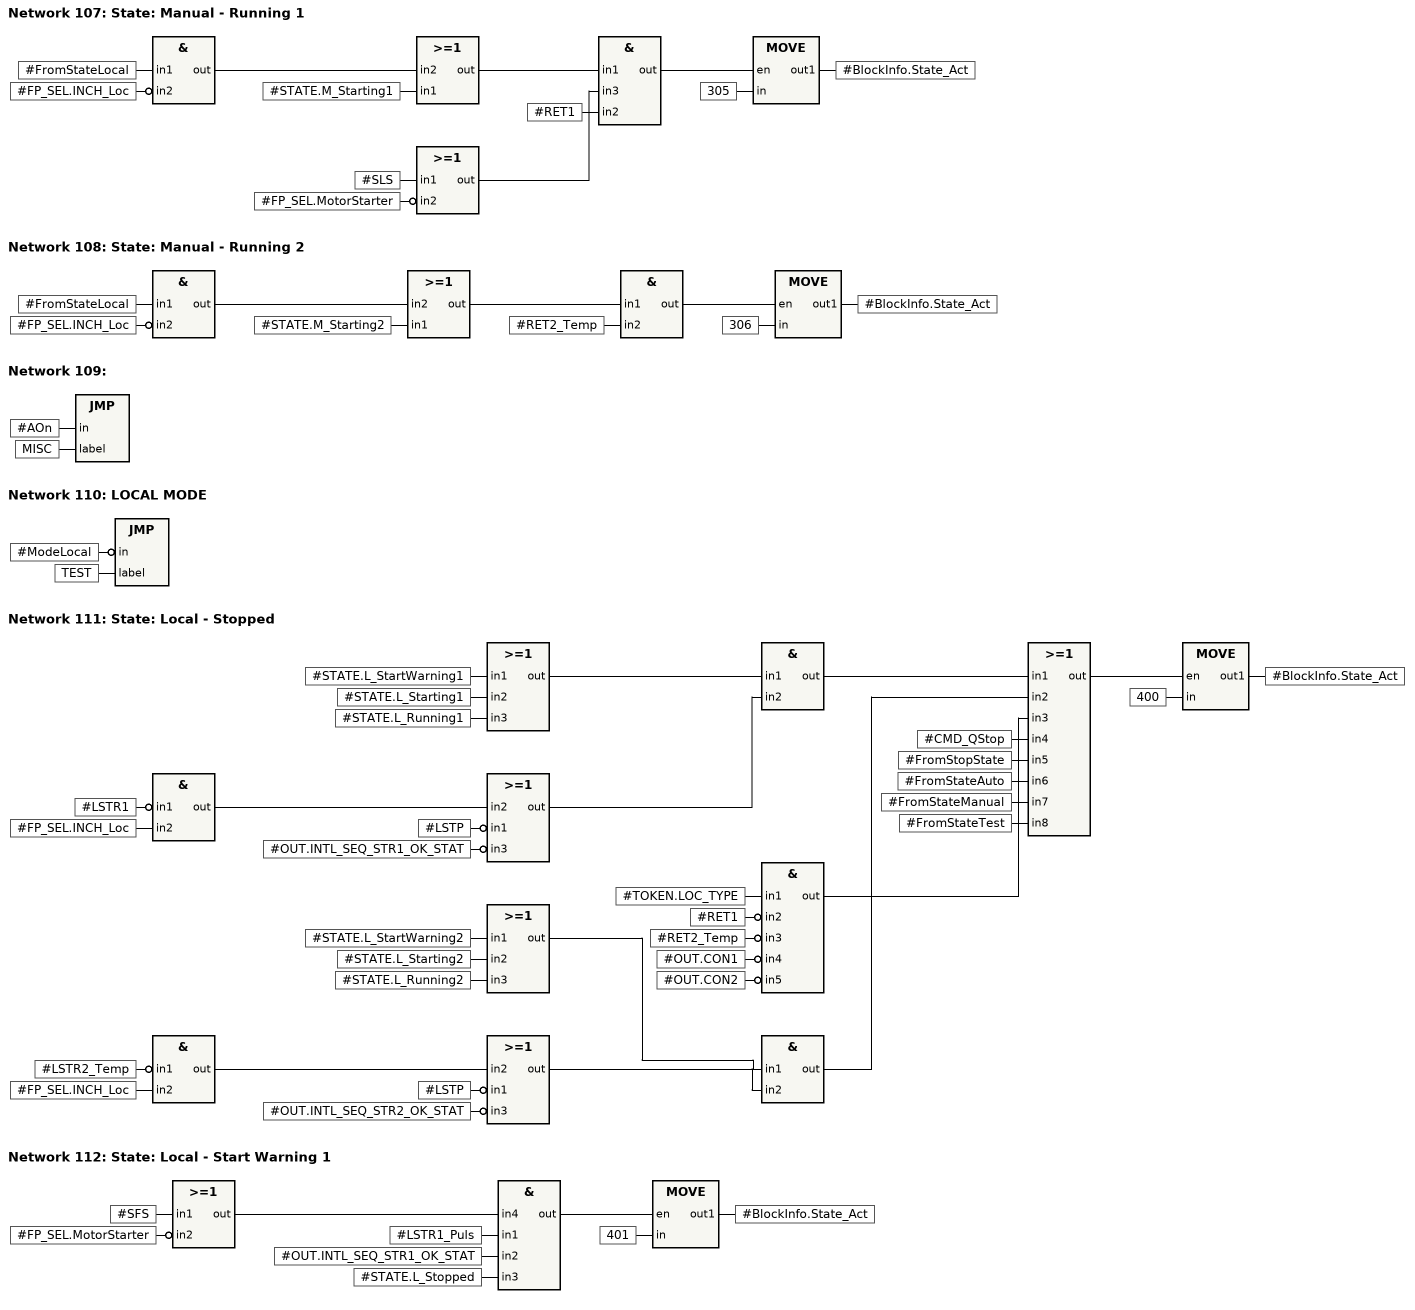
   IF ((#FromStateLocal AND NOT #FP_SEL.INCH_Loc) OR #STATE.M_Starting1) AND (#SLS OR NOT #FP_SEL.MotorStarter) AND #RET1 THEN
       #BlockInfo.State_Act := 305;
   END_IF;
END_REGION

REGION Network 108: State: Manual - Running 2
   IF ((#FromStateLocal AND NOT #FP_SEL.INCH_Loc) OR #STATE.M_Starting2) AND #RET2_Temp THEN
       #BlockInfo.State_Act := 306;
   END_IF;
END_REGION

REGION Network 109
   IF #AOn THEN GOTO MISC; END_IF;
END_REGION

REGION Network 110: LOCAL MODE
   LOC:
   IF NOT #ModeLocal THEN GOTO TEST; END_IF;
END_REGION

REGION Network 111: State: Local - Stopped
   IF ((#STATE.L_StartWarning1 OR #STATE.L_Starting1 OR #STATE.L_Running1) AND ((NOT #LSTR1 AND #FP_SEL.INCH_Loc) OR NOT #LSTP OR NOT #OUT.INTL_SEQ_STR1_OK_STAT)) OR ((#STATE.L_StartWarning2 OR #STATE.L_Starting2 OR #STATE.L_Running2) AND ((NOT #LSTR2_Temp AND #FP_SEL.INCH_Loc) OR NOT #LSTP OR NOT #OUT.INTL_SEQ_STR2_OK_STAT)) OR (#TOKEN.LOC_TYPE AND NOT #RET1 AND NOT #RET2_Temp AND NOT #OUT.CON1 AND NOT #OUT.CON2) OR #CMD_QStop OR #FromStopState OR #FromStateAuto OR #FromStateManual OR #FromStateTest THEN
       #BlockInfo.State_Act := 400;
   END_IF;
END_REGION

REGION Network 112: State: Local - Start Warning 1
   IF (#SFS OR NOT #FP_SEL.MotorStarter) AND #LSTR1_Puls AND #OUT.INTL_SEQ_STR1_OK_STAT AND #STATE.L_Stopped THEN
       #BlockInfo.State_Act := 401;
   END_IF;
END_REGION

REGION Network 113: State: Local - Start Warning 2
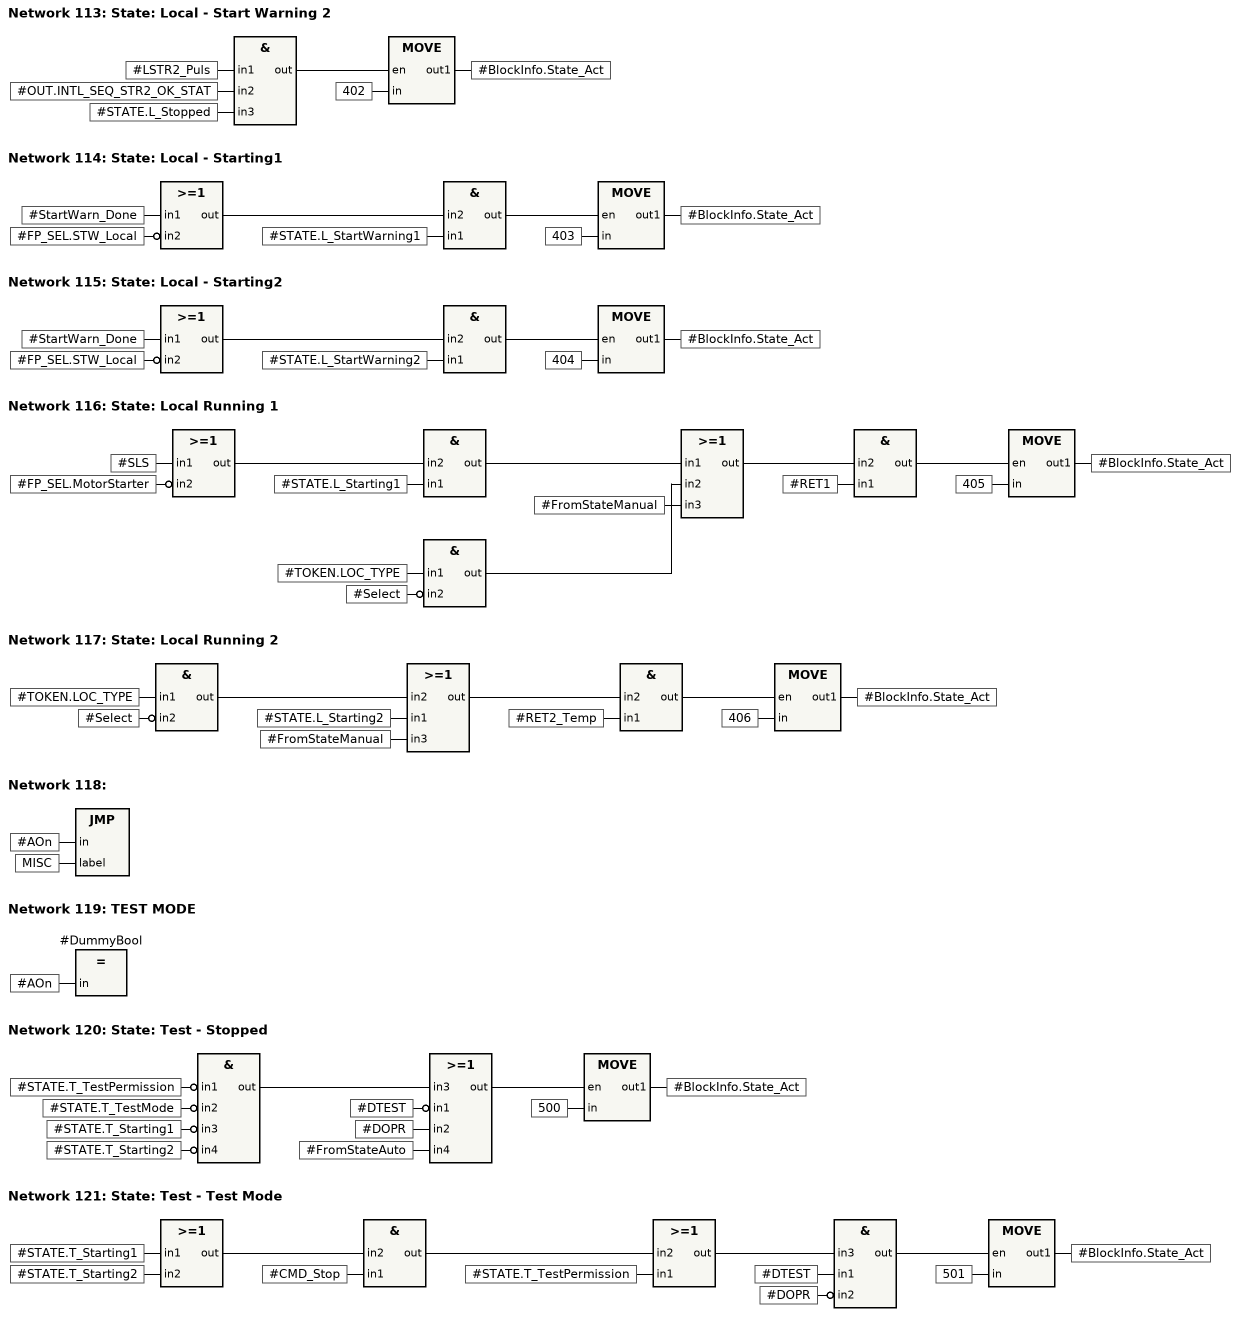
   IF #LSTR2_Puls AND #OUT.INTL_SEQ_STR2_OK_STAT AND #STATE.L_Stopped THEN
       #BlockInfo.State_Act := 402;
   END_IF;
END_REGION

REGION Network 114: State: Local - Starting1
   IF (#StartWarn_Done OR NOT #FP_SEL.STW_Local) AND #STATE.L_StartWarning1 THEN
       #BlockInfo.State_Act := 403;
   END_IF;
END_REGION

REGION Network 115: State: Local - Starting2
   IF (#StartWarn_Done OR NOT #FP_SEL.STW_Local) AND #STATE.L_StartWarning2 THEN
       #BlockInfo.State_Act := 404;
   END_IF;
END_REGION

REGION Network 116: State: Local Running 1
   IF (((#SLS OR NOT #FP_SEL.MotorStarter) AND #STATE.L_Starting1) OR (#TOKEN.LOC_TYPE AND NOT #Select) OR #FromStateManual) AND #RET1 THEN
       #BlockInfo.State_Act := 405;
   END_IF;
END_REGION

REGION Network 117: State: Local Running 2
   IF ((#TOKEN.LOC_TYPE AND NOT #Select) OR #STATE.L_Starting2 OR #FromStateManual) AND #RET2_Temp THEN
       #BlockInfo.State_Act := 406;
   END_IF;
END_REGION

REGION Network 118
   IF #AOn THEN GOTO MISC; END_IF;
END_REGION

REGION Network 119: TEST MODE
   TEST:
   #DummyBool := #AOn;
END_REGION

REGION Network 120: State: Test - Stopped
   IF (NOT #STATE.T_TestPermission AND NOT #STATE.T_TestMode AND NOT #STATE.T_Starting1 AND NOT #STATE.T_Starting2) OR NOT #DTEST OR #DOPR OR #FromStateAuto THEN
       #BlockInfo.State_Act := 500;
   END_IF;
END_REGION

REGION Network 121: State: Test - Test Mode
   IF (((#STATE.T_Starting1 OR #STATE.T_Starting2) AND #CMD_Stop) OR #STATE.T_TestPermission) AND #DTEST AND NOT #DOPR THEN
       #BlockInfo.State_Act := 501;
   END_IF;
END_REGION

REGION Network 122: State: Test - Starting 1
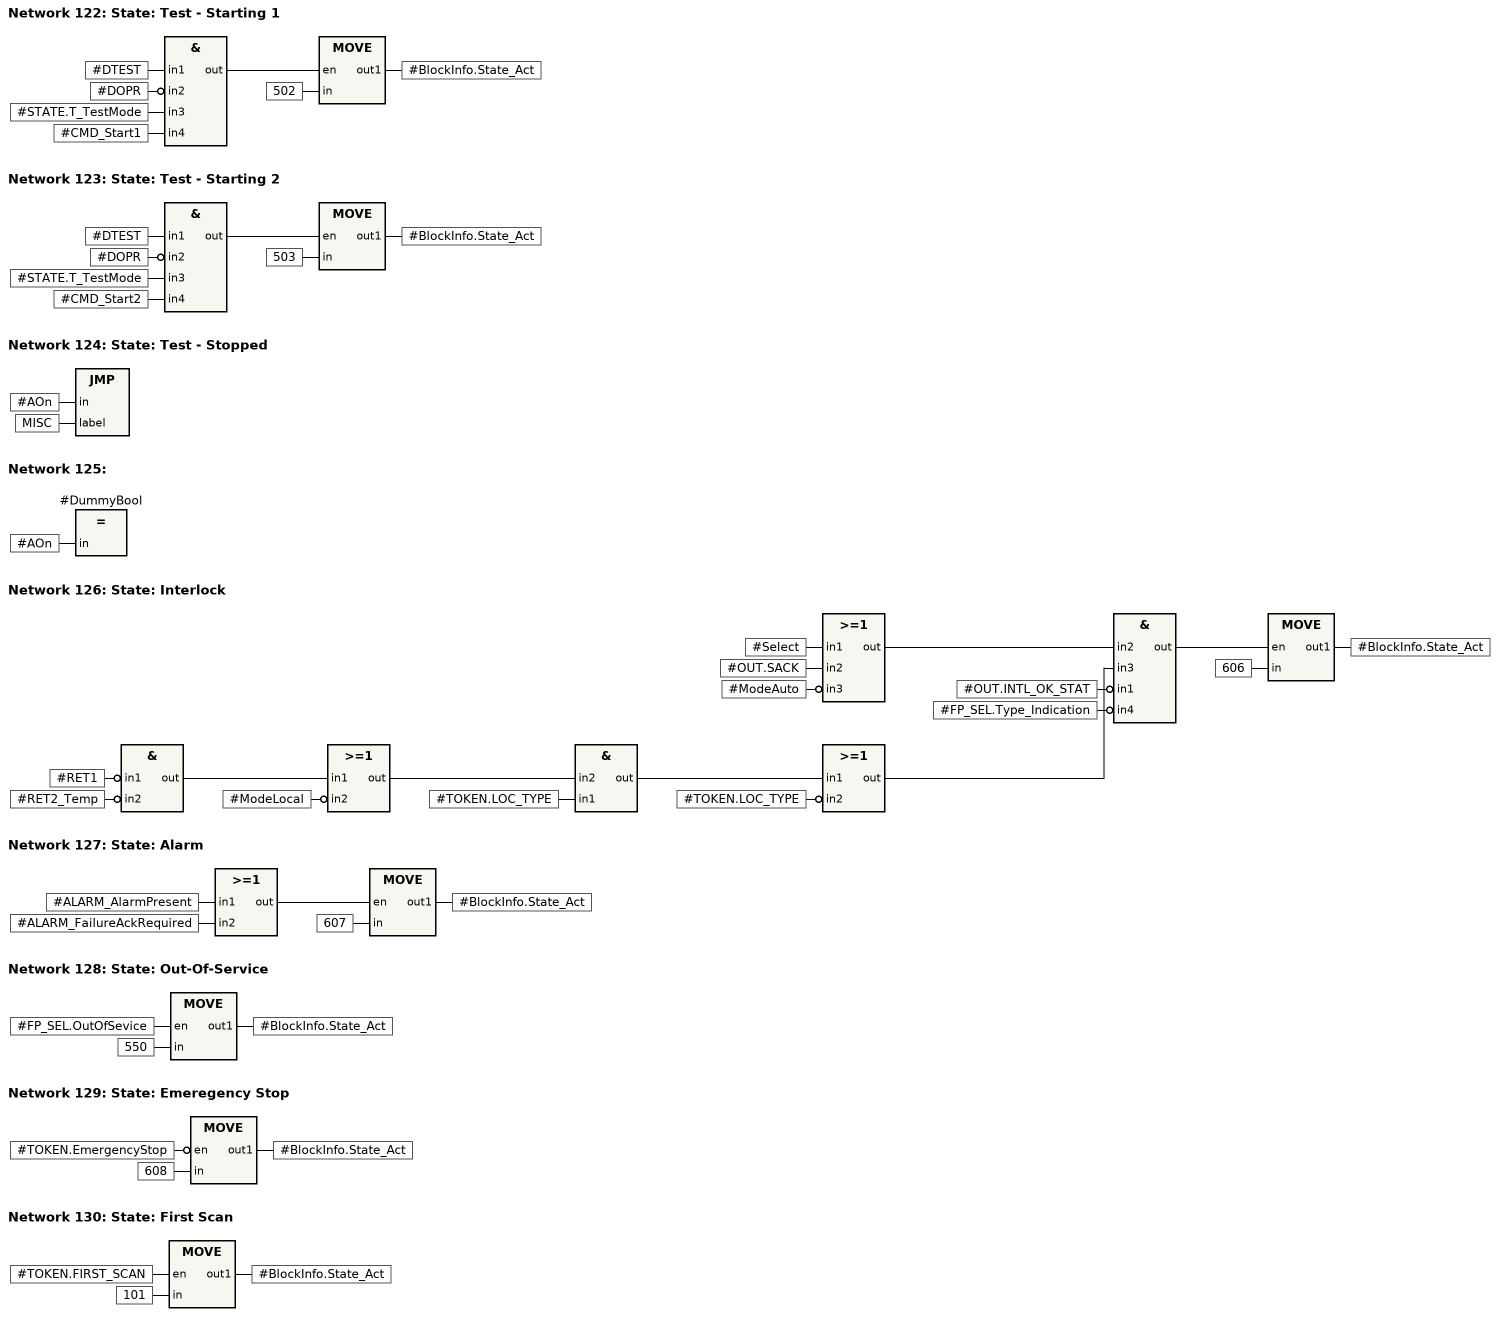
   IF #DTEST AND NOT #DOPR AND #STATE.T_TestMode AND #CMD_Start1 THEN #BlockInfo.State_Act := 502; END_IF;
END_REGION

REGION Network 123: State: Test - Starting 2
   IF #DTEST AND NOT #DOPR AND #STATE.T_TestMode AND #CMD_Start2 THEN #BlockInfo.State_Act := 503; END_IF;
END_REGION

REGION Network 124: State: Test - Stopped
   IF #AOn THEN GOTO MISC; END_IF;
END_REGION

REGION Network 125
   MISC:
   #DummyBool := #AOn;
END_REGION

REGION Network 126: State: Interlock
   // Build 007 - 06 Feb 2020 (EXTBOB) : FP_SEL Indication negate added to Interlock state
   IF (#Select OR #OUT.SACK OR NOT #ModeAuto) AND ((((NOT #RET1 AND NOT #RET2_Temp) OR NOT #ModeLocal) AND #TOKEN.LOC_TYPE) OR NOT #TOKEN.LOC_TYPE) AND NOT #OUT.INTL_OK_STAT AND NOT #FP_SEL.Type_Indication THEN
       #BlockInfo.State_Act := 606;
   END_IF;
END_REGION

REGION Network 127: State: Alarm
   IF #ALARM_AlarmPresent OR #ALARM_FailureAckRequired THEN #BlockInfo.State_Act := 607; END_IF;
END_REGION

REGION Network 128: State: Out-Of-Service
   IF #FP_SEL.OutOfSevice THEN #BlockInfo.State_Act := 550; END_IF;
END_REGION

REGION Network 129: State: Emeregency Stop
   IF NOT #TOKEN.EmergencyStop THEN #BlockInfo.State_Act := 608; END_IF;
END_REGION

REGION Network 130: State: First Scan
   IF #TOKEN.FIRST_SCAN THEN #BlockInfo.State_Act := 101; END_IF;
END_REGION

REGION Network 131: State: Stopped1
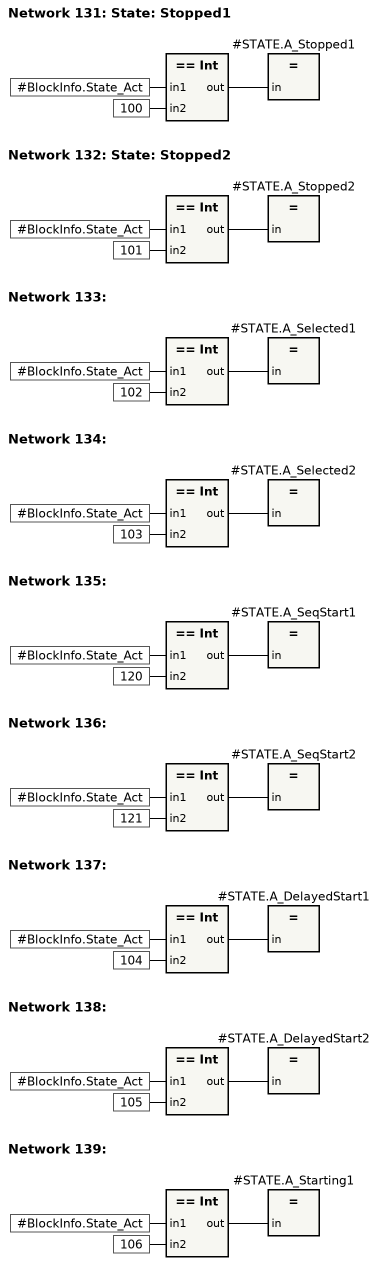
   #STATE.A_Stopped1 := #BlockInfo.State_Act = 100;
END_REGION

REGION Network 132: State: Stopped2
   #STATE.A_Stopped2 := #BlockInfo.State_Act = 101;
END_REGION

REGION Network 133
   #STATE.A_Selected1 := #BlockInfo.State_Act = 102;
END_REGION

REGION Network 134
   #STATE.A_Selected2 := #BlockInfo.State_Act = 103;
END_REGION

REGION Network 135
   #STATE.A_SeqStart1 := #BlockInfo.State_Act = 120;
END_REGION

REGION Network 136
   #STATE.A_SeqStart2 := #BlockInfo.State_Act = 121;
END_REGION

REGION Network 137
   #STATE.A_DelayedStart1 := #BlockInfo.State_Act = 104;
END_REGION

REGION Network 138
   #STATE.A_DelayedStart2 := #BlockInfo.State_Act = 105;
END_REGION

REGION Network 139
   #STATE.A_Starting1 := #BlockInfo.State_Act = 106;
END_REGION

REGION Network 140
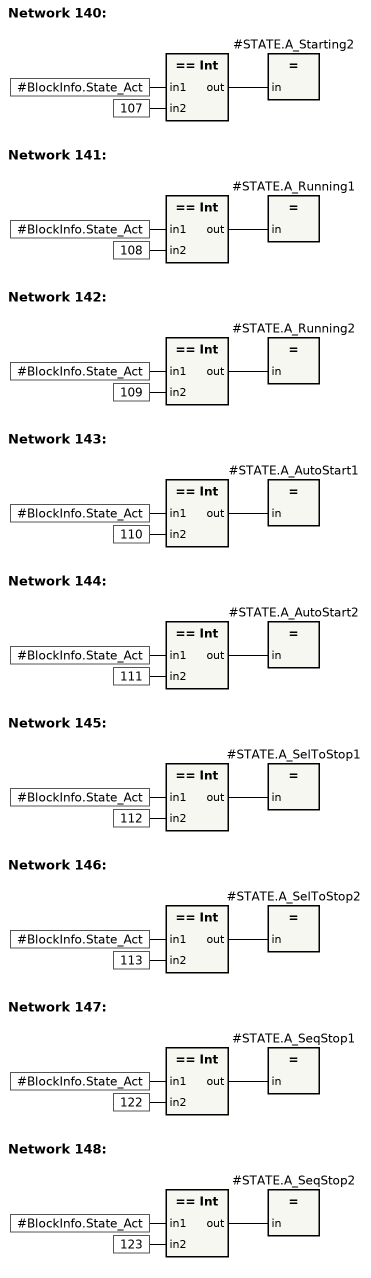
   #STATE.A_Starting2 := #BlockInfo.State_Act = 107;
END_REGION

REGION Network 141
   #STATE.A_Running1 := #BlockInfo.State_Act = 108;
END_REGION

REGION Network 142
   #STATE.A_Running2 := #BlockInfo.State_Act = 109;
END_REGION

REGION Network 143
   #STATE.A_AutoStart1 := #BlockInfo.State_Act = 110;
END_REGION

REGION Network 144
   #STATE.A_AutoStart2 := #BlockInfo.State_Act = 111;
END_REGION

REGION Network 145
   #STATE.A_SelToStop1 := #BlockInfo.State_Act = 112;
END_REGION

REGION Network 146
   #STATE.A_SelToStop2 := #BlockInfo.State_Act = 113;
END_REGION

REGION Network 147
   #STATE.A_SeqStop1 := #BlockInfo.State_Act = 122;
END_REGION

REGION Network 148
   #STATE.A_SeqStop2 := #BlockInfo.State_Act = 123;
END_REGION

REGION Network 149
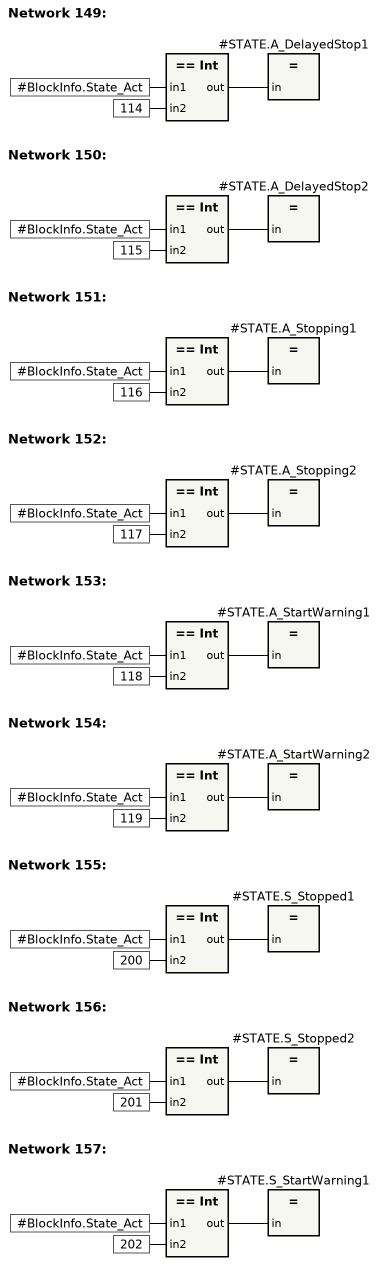
   #STATE.A_DelayedStop1 := #BlockInfo.State_Act = 114;
END_REGION

REGION Network 150
   #STATE.A_DelayedStop2 := #BlockInfo.State_Act = 115;
END_REGION

REGION Network 151
   #STATE.A_Stopping1 := #BlockInfo.State_Act = 116;
END_REGION

REGION Network 152
   #STATE.A_Stopping2 := #BlockInfo.State_Act = 117;
END_REGION

REGION Network 153
   #STATE.A_StartWarning1 := #BlockInfo.State_Act = 118;
END_REGION

REGION Network 154
   #STATE.A_StartWarning2 := #BlockInfo.State_Act = 119;
END_REGION

REGION Network 155
   #STATE.S_Stopped1 := #BlockInfo.State_Act = 200;
END_REGION

REGION Network 156
   #STATE.S_Stopped2 := #BlockInfo.State_Act = 201;
END_REGION

REGION Network 157
   #STATE.S_StartWarning1 := #BlockInfo.State_Act = 202;
END_REGION

REGION Network 158
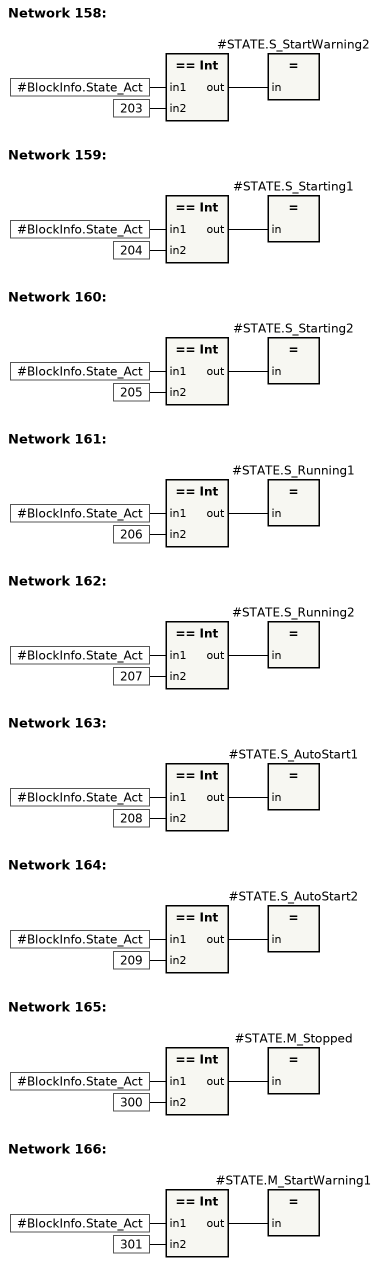
   #STATE.S_StartWarning2 := #BlockInfo.State_Act = 203;
END_REGION

REGION Network 159
   #STATE.S_Starting1 := #BlockInfo.State_Act = 204;
END_REGION

REGION Network 160
   #STATE.S_Starting2 := #BlockInfo.State_Act = 205;
END_REGION

REGION Network 161
   #STATE.S_Running1 := #BlockInfo.State_Act = 206;
END_REGION

REGION Network 162
   #STATE.S_Running2 := #BlockInfo.State_Act = 207;
END_REGION

REGION Network 163
   #STATE.S_AutoStart1 := #BlockInfo.State_Act = 208;
END_REGION

REGION Network 164
   #STATE.S_AutoStart2 := #BlockInfo.State_Act = 209;
END_REGION

REGION Network 165
   #STATE.M_Stopped := #BlockInfo.State_Act = 300;
END_REGION

REGION Network 166
   #STATE.M_StartWarning1 := #BlockInfo.State_Act = 301;
END_REGION

REGION Network 167
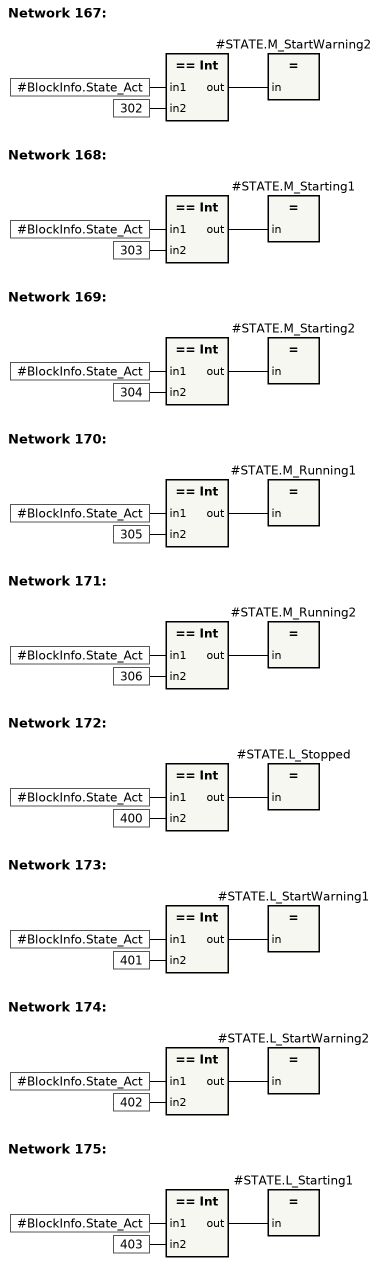
   #STATE.M_StartWarning2 := #BlockInfo.State_Act = 302;
END_REGION

REGION Network 168
   #STATE.M_Starting1 := #BlockInfo.State_Act = 303;
END_REGION

REGION Network 169
   #STATE.M_Starting2 := #BlockInfo.State_Act = 304;
END_REGION

REGION Network 170
   #STATE.M_Running1 := #BlockInfo.State_Act = 305;
END_REGION

REGION Network 171
   #STATE.M_Running2 := #BlockInfo.State_Act = 306;
END_REGION

REGION Network 172
   #STATE.L_Stopped := #BlockInfo.State_Act = 400;
END_REGION

REGION Network 173
   #STATE.L_StartWarning1 := #BlockInfo.State_Act = 401;
END_REGION

REGION Network 174
   #STATE.L_StartWarning2 := #BlockInfo.State_Act = 402;
END_REGION

REGION Network 175
   #STATE.L_Starting1 := #BlockInfo.State_Act = 403;
END_REGION

REGION Network 176
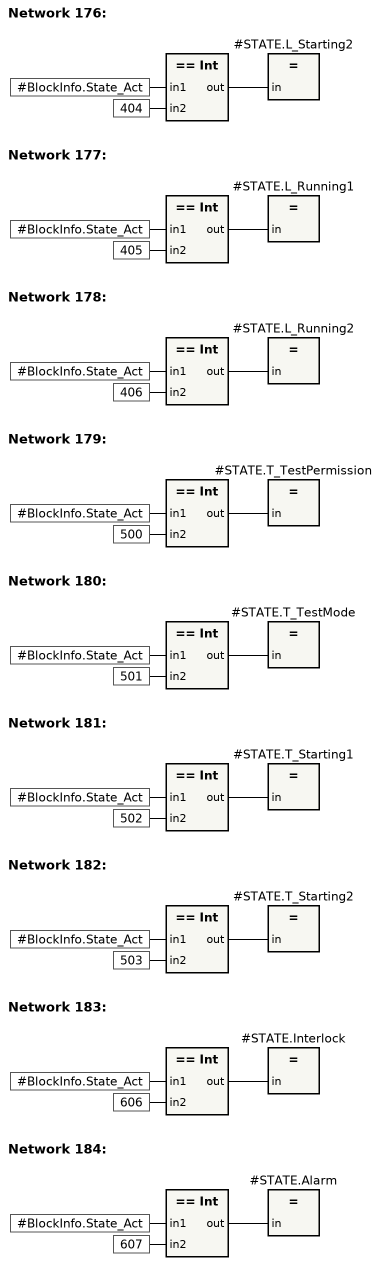
   #STATE.L_Starting2 := #BlockInfo.State_Act = 404;
END_REGION

REGION Network 177
   #STATE.L_Running1 := #BlockInfo.State_Act = 405;
END_REGION

REGION Network 178
   #STATE.L_Running2 := #BlockInfo.State_Act = 406;
END_REGION

REGION Network 179
   #STATE.T_TestPermission := #BlockInfo.State_Act = 500;
END_REGION

REGION Network 180
   #STATE.T_TestMode := #BlockInfo.State_Act = 501;
END_REGION

REGION Network 181
   #STATE.T_Starting1 := #BlockInfo.State_Act = 502;
END_REGION

REGION Network 182
   #STATE.T_Starting2 := #BlockInfo.State_Act = 503;
END_REGION

REGION Network 183
   #STATE.Interlock := #BlockInfo.State_Act = 606;
END_REGION

REGION Network 184
   #STATE.Alarm := #BlockInfo.State_Act = 607;
END_REGION

REGION Network 185
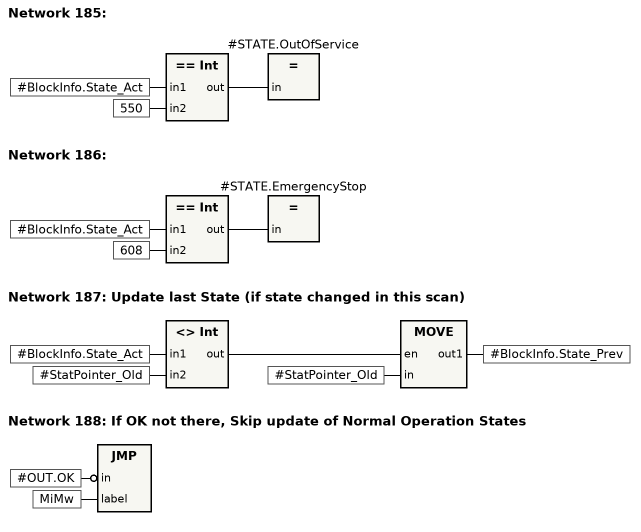
   #STATE.OutOfService := #BlockInfo.State_Act = 550;
END_REGION

REGION Network 186
   #STATE.EmergencyStop := #BlockInfo.State_Act = 608;
END_REGION

REGION Network 187: Update last State (if state changed in this scan)
   IF #BlockInfo.State_Act <> #StatPointer_Old THEN #BlockInfo.State_Prev := #StatPointer_Old; END_IF;
END_REGION

REGION Network 188: If OK not there, Skip update of Normal Operation States
   // Build 010 - 30.09.2020 (EXTBOB): Skipped Normal MSW status update in case of Alarm Condition, Newly Added
   IF NOT #OUT.OK THEN GOTO MiMw; END_IF;
END_REGION

REGION Network 189: UPDATE MSW
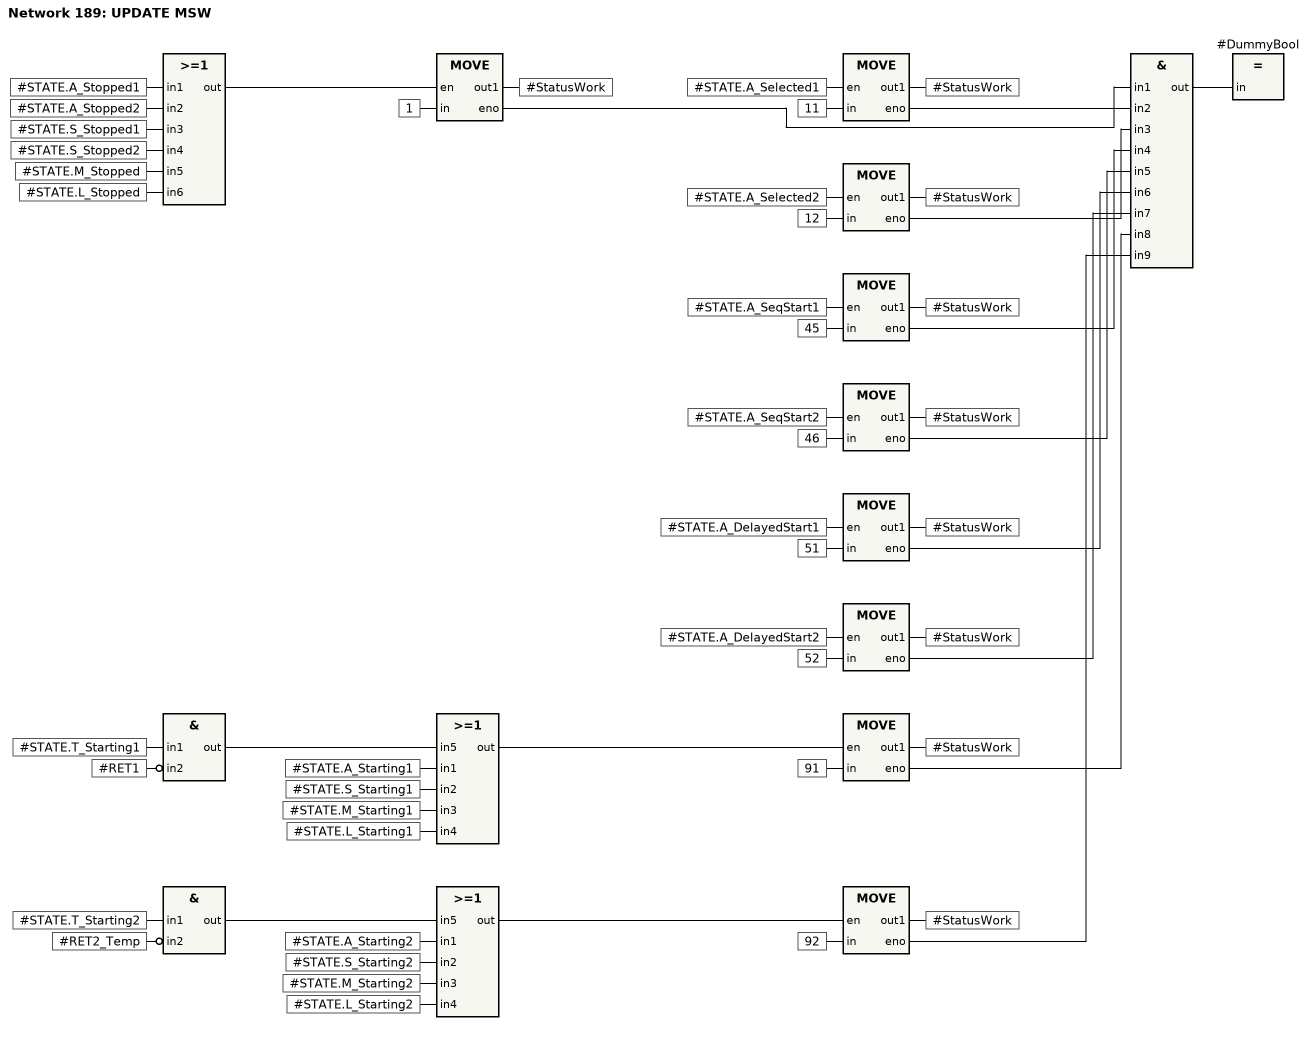
   // ENO of a box is taken as its EN; it also drops when the box reports an error
   #_w1 := #STATE.A_Stopped1 OR #STATE.A_Stopped2 OR #STATE.S_Stopped1 OR #STATE.S_Stopped2 OR #STATE.M_Stopped OR #STATE.L_Stopped;
   IF #_w1 THEN #StatusWork := 1; END_IF;
   IF #STATE.A_Selected1 THEN #StatusWork := 11; END_IF;
   IF #STATE.A_Selected2 THEN #StatusWork := 12; END_IF;
   IF #STATE.A_SeqStart1 THEN #StatusWork := 45; END_IF;
   IF #STATE.A_SeqStart2 THEN #StatusWork := 46; END_IF;
   IF #STATE.A_DelayedStart1 THEN #StatusWork := 51; END_IF;
   IF #STATE.A_DelayedStart2 THEN #StatusWork := 52; END_IF;
   #_w2 := (#STATE.T_Starting1 AND NOT #RET1) OR #STATE.A_Starting1 OR #STATE.S_Starting1 OR #STATE.M_Starting1 OR #STATE.L_Starting1;
   IF #_w2 THEN #StatusWork := 91; END_IF;
   #_w3 := (#STATE.T_Starting2 AND NOT #RET2_Temp) OR #STATE.A_Starting2 OR #STATE.S_Starting2 OR #STATE.M_Starting2 OR #STATE.L_Starting2;
   IF #_w3 THEN #StatusWork := 92; END_IF;
   #DummyBool := #_w1 AND #STATE.A_Selected1 AND #STATE.A_Selected2 AND #STATE.A_SeqStart1 AND #STATE.A_SeqStart2 AND #STATE.A_DelayedStart1 AND #STATE.A_DelayedStart2 AND #_w2 AND #_w3;
END_REGION

REGION Network 190
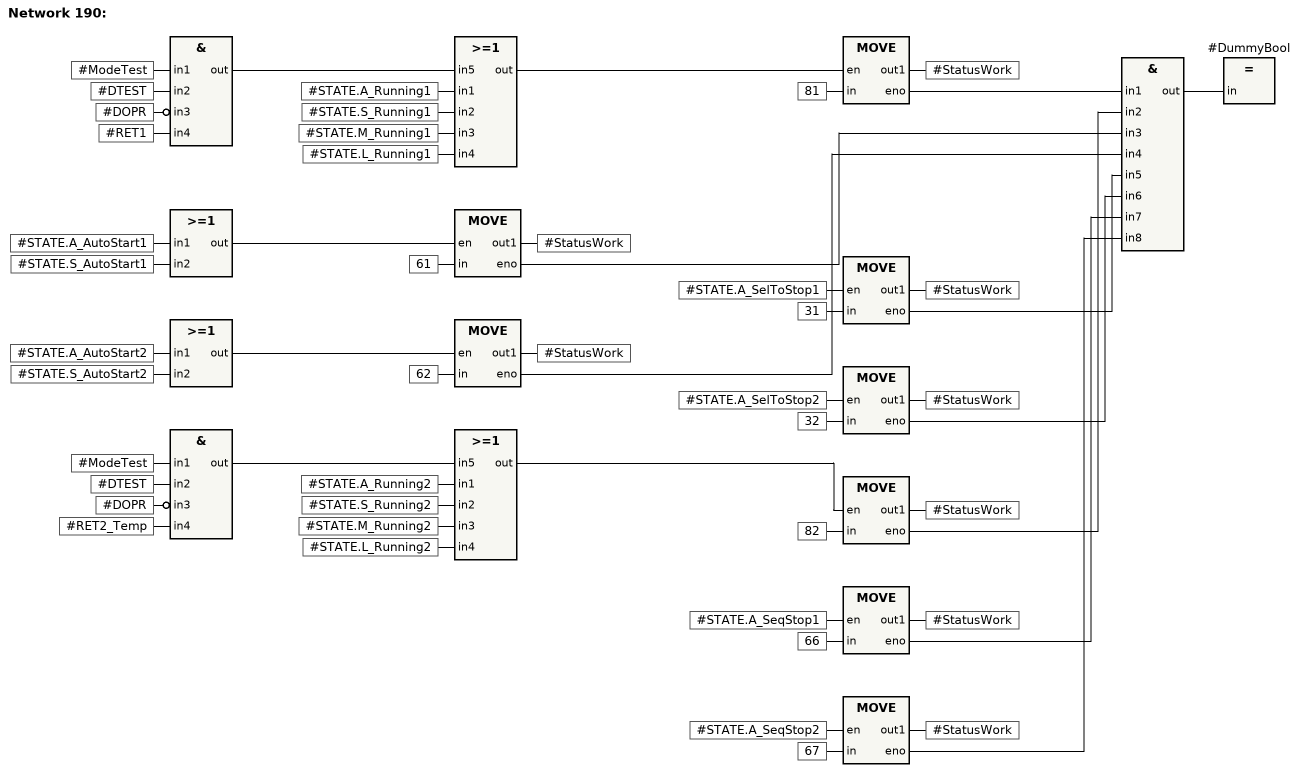
   // ENO of a box is taken as its EN; it also drops when the box reports an error
   #_w1 := (#ModeTest AND #DTEST AND NOT #DOPR AND #RET1) OR #STATE.A_Running1 OR #STATE.S_Running1 OR #STATE.M_Running1 OR #STATE.L_Running1;
   IF #_w1 THEN #StatusWork := 81; END_IF;
   #_w2 := (#ModeTest AND #DTEST AND NOT #DOPR AND #RET2_Temp) OR #STATE.A_Running2 OR #STATE.S_Running2 OR #STATE.M_Running2 OR #STATE.L_Running2;
   IF #_w2 THEN #StatusWork := 82; END_IF;
   #_w3 := #STATE.A_AutoStart1 OR #STATE.S_AutoStart1;
   IF #_w3 THEN #StatusWork := 61; END_IF;
   #_w4 := #STATE.A_AutoStart2 OR #STATE.S_AutoStart2;
   IF #_w4 THEN #StatusWork := 62; END_IF;
   IF #STATE.A_SelToStop1 THEN #StatusWork := 31; END_IF;
   IF #STATE.A_SelToStop2 THEN #StatusWork := 32; END_IF;
   IF #STATE.A_SeqStop1 THEN #StatusWork := 66; END_IF;
   IF #STATE.A_SeqStop2 THEN #StatusWork := 67; END_IF;
   #DummyBool := #_w1 AND #_w2 AND #_w3 AND #_w4 AND #STATE.A_SelToStop1 AND #STATE.A_SelToStop2 AND #STATE.A_SeqStop1 AND #STATE.A_SeqStop2;
END_REGION

REGION Network 191
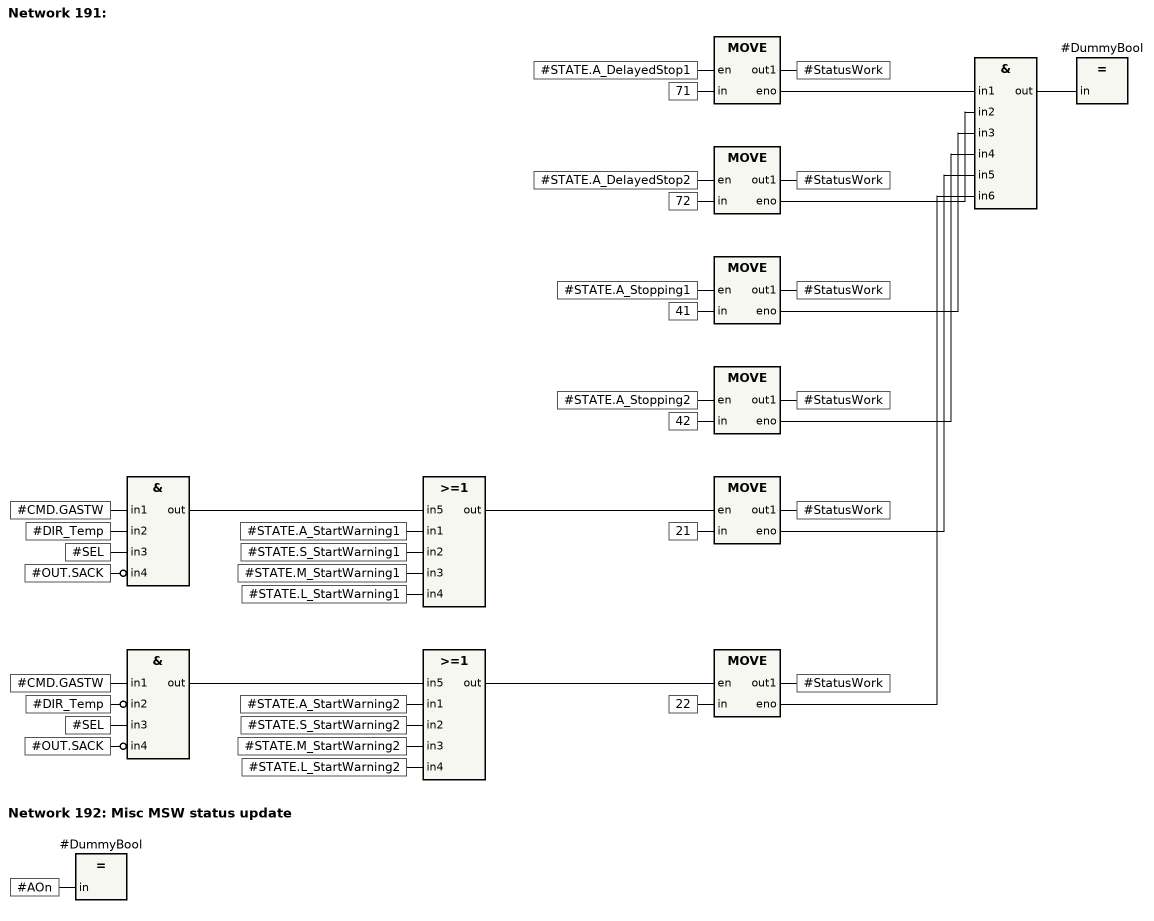
   // ENO of a box is taken as its EN; it also drops when the box reports an error
   IF #STATE.A_DelayedStop1 THEN #StatusWork := 71; END_IF;
   IF #STATE.A_DelayedStop2 THEN #StatusWork := 72; END_IF;
   IF #STATE.A_Stopping1 THEN #StatusWork := 41; END_IF;
   IF #STATE.A_Stopping2 THEN #StatusWork := 42; END_IF;
   #_w1 := (#CMD.GASTW AND #DIR_Temp AND #SEL AND NOT #OUT.SACK) OR #STATE.A_StartWarning1 OR #STATE.S_StartWarning1 OR #STATE.M_StartWarning1 OR #STATE.L_StartWarning1;
   IF #_w1 THEN #StatusWork := 21; END_IF;
   #_w2 := (#CMD.GASTW AND NOT #DIR_Temp AND #SEL AND NOT #OUT.SACK) OR #STATE.A_StartWarning2 OR #STATE.S_StartWarning2 OR #STATE.M_StartWarning2 OR #STATE.L_StartWarning2;
   IF #_w2 THEN #StatusWork := 22; END_IF;
   #DummyBool := #STATE.A_DelayedStop1 AND #STATE.A_DelayedStop2 AND #STATE.A_Stopping1 AND #STATE.A_Stopping2 AND #_w1 AND #_w2;
END_REGION

REGION Network 192: Misc MSW status update
   // Build 010 - 30.09.2020 (EXTBOB): Skipped Normal MSW status update in case of Alarm Condition, Newly Added
   MiMw:
   #DummyBool := #AOn;
END_REGION

REGION Network 193
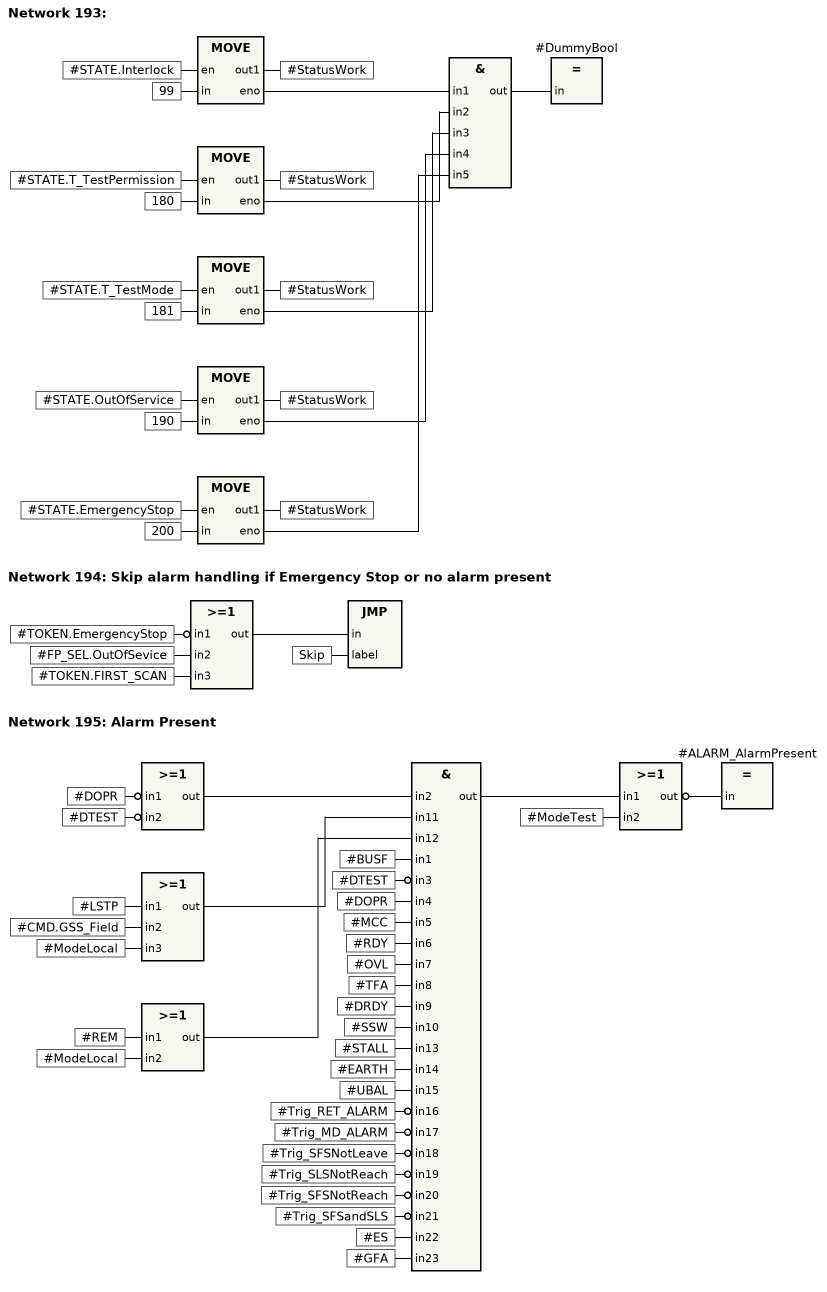
   // ENO of a box is taken as its EN; it also drops when the box reports an error
   IF #STATE.Interlock THEN #StatusWork := 99; END_IF;
   IF #STATE.T_TestPermission THEN #StatusWork := 180; END_IF;
   IF #STATE.T_TestMode THEN #StatusWork := 181; END_IF;
   IF #STATE.OutOfService THEN #StatusWork := 190; END_IF;
   IF #STATE.EmergencyStop THEN #StatusWork := 200; END_IF;
   #DummyBool := #STATE.Interlock AND #STATE.T_TestPermission AND #STATE.T_TestMode AND #STATE.OutOfService AND #STATE.EmergencyStop;
END_REGION

REGION Network 194: Skip alarm handling if Emergency Stop or no alarm present
   // Skip = Skip Alarm
   IF NOT #TOKEN.EmergencyStop OR #FP_SEL.OutOfSevice OR #TOKEN.FIRST_SCAN THEN GOTO Skip; END_IF;
END_REGION

REGION Network 195: Alarm Present
   #ALARM_AlarmPresent := NOT (((NOT #DOPR OR NOT #DTEST) AND (#LSTP OR #CMD.GSS_Field OR #ModeLocal) AND (#REM OR #ModeLocal) AND #BUSF AND NOT #DTEST AND #DOPR AND #MCC AND #RDY AND #OVL AND #TFA AND #DRDY AND #SSW AND #STALL AND #EARTH AND #UBAL AND NOT #Trig_RET_ALARM AND NOT #Trig_MD_ALARM AND NOT #Trig_SFSNotLeave AND NOT #Trig_SLSNotReach AND NOT #Trig_SFSNotReach AND NOT #Trig_SFSandSLS AND #ES AND #GFA) OR #ModeTest);
END_REGION

REGION Network 196
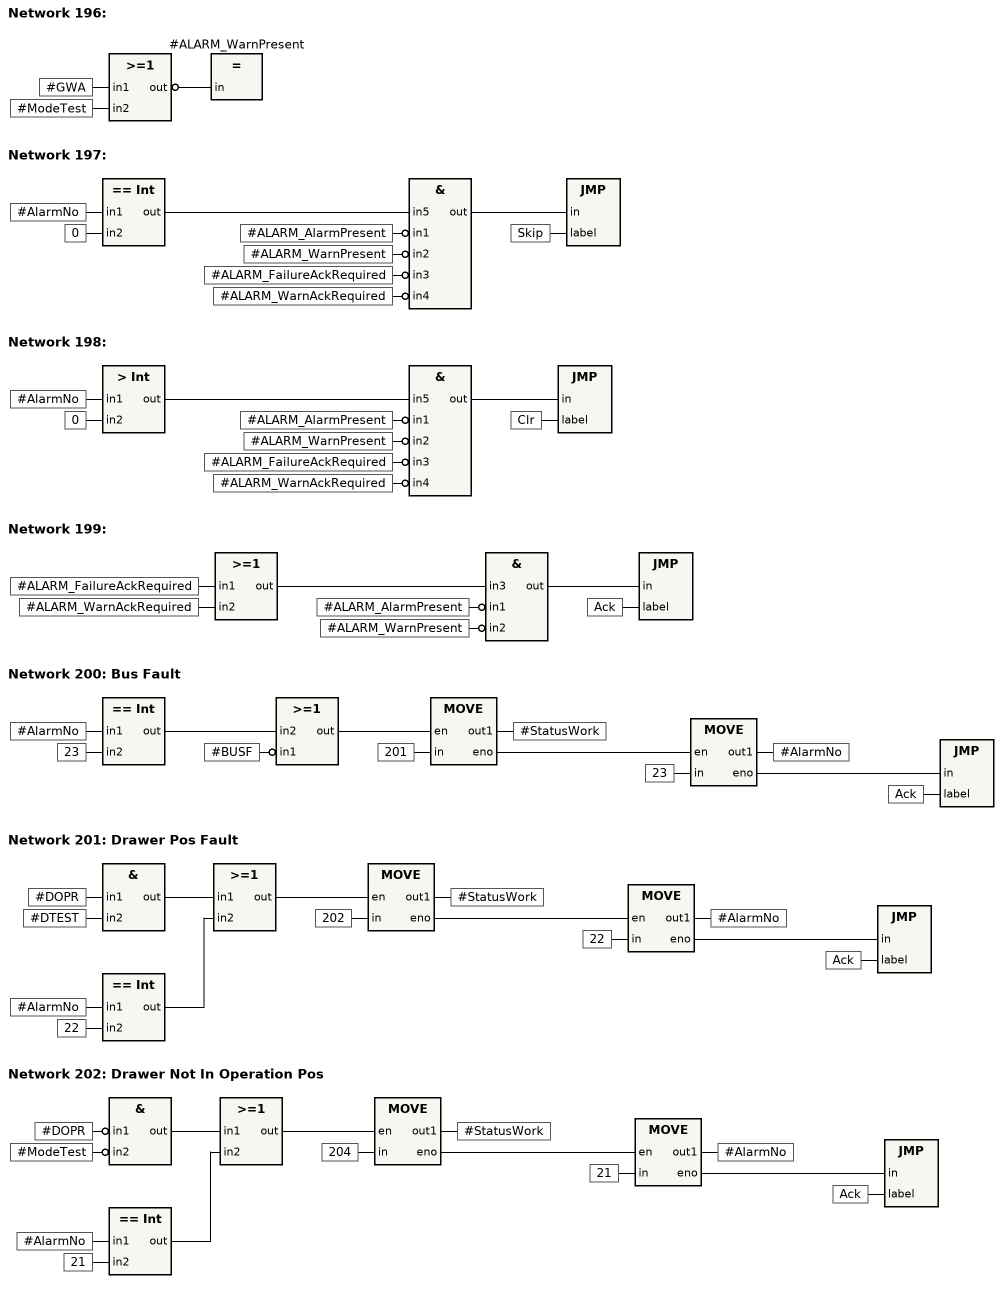
   #ALARM_WarnPresent := NOT (#GWA OR #ModeTest);
END_REGION

REGION Network 197
   // Skip = Skip Alarm
   IF (#AlarmNo = 0) AND NOT #ALARM_AlarmPresent AND NOT #ALARM_WarnPresent AND NOT #ALARM_FailureAckRequired AND NOT #ALARM_WarnAckRequired THEN
       GOTO Skip;
   END_IF;
END_REGION

REGION Network 198
   // Clr = Clear Alarm
   IF (#AlarmNo > 0) AND NOT #ALARM_AlarmPresent AND NOT #ALARM_WarnPresent AND NOT #ALARM_FailureAckRequired AND NOT #ALARM_WarnAckRequired THEN
       GOTO Clr;
   END_IF;
END_REGION

REGION Network 199
   // Ack = Alarm Acknowledge
   IF (#ALARM_FailureAckRequired OR #ALARM_WarnAckRequired) AND NOT #ALARM_AlarmPresent AND NOT #ALARM_WarnPresent THEN
       GOTO Ack;
   END_IF;
END_REGION

REGION Network 200: Bus Fault
   // ENO of a box is taken as its EN; it also drops when the box reports an error
   #_w1 := (#AlarmNo = 23) OR NOT #BUSF;
   IF #_w1 THEN
       #StatusWork := 201;
       #AlarmNo := 23;
       GOTO Ack;
   END_IF;
END_REGION

REGION Network 201: Drawer Pos Fault
   // ENO of a box is taken as its EN; it also drops when the box reports an error
   #_w1 := (#DOPR AND #DTEST) OR (#AlarmNo = 22);
   IF #_w1 THEN
       #StatusWork := 202;
       #AlarmNo := 22;
       GOTO Ack;
   END_IF;
END_REGION

REGION Network 202: Drawer Not In Operation Pos
   // ENO of a box is taken as its EN; it also drops when the box reports an error
   #_w1 := (NOT #DOPR AND NOT #ModeTest) OR (#AlarmNo = 21);
   IF #_w1 THEN
       #StatusWork := 204;
       #AlarmNo := 21;
       GOTO Ack;
   END_IF;
END_REGION

REGION Network 203: MCC Fault
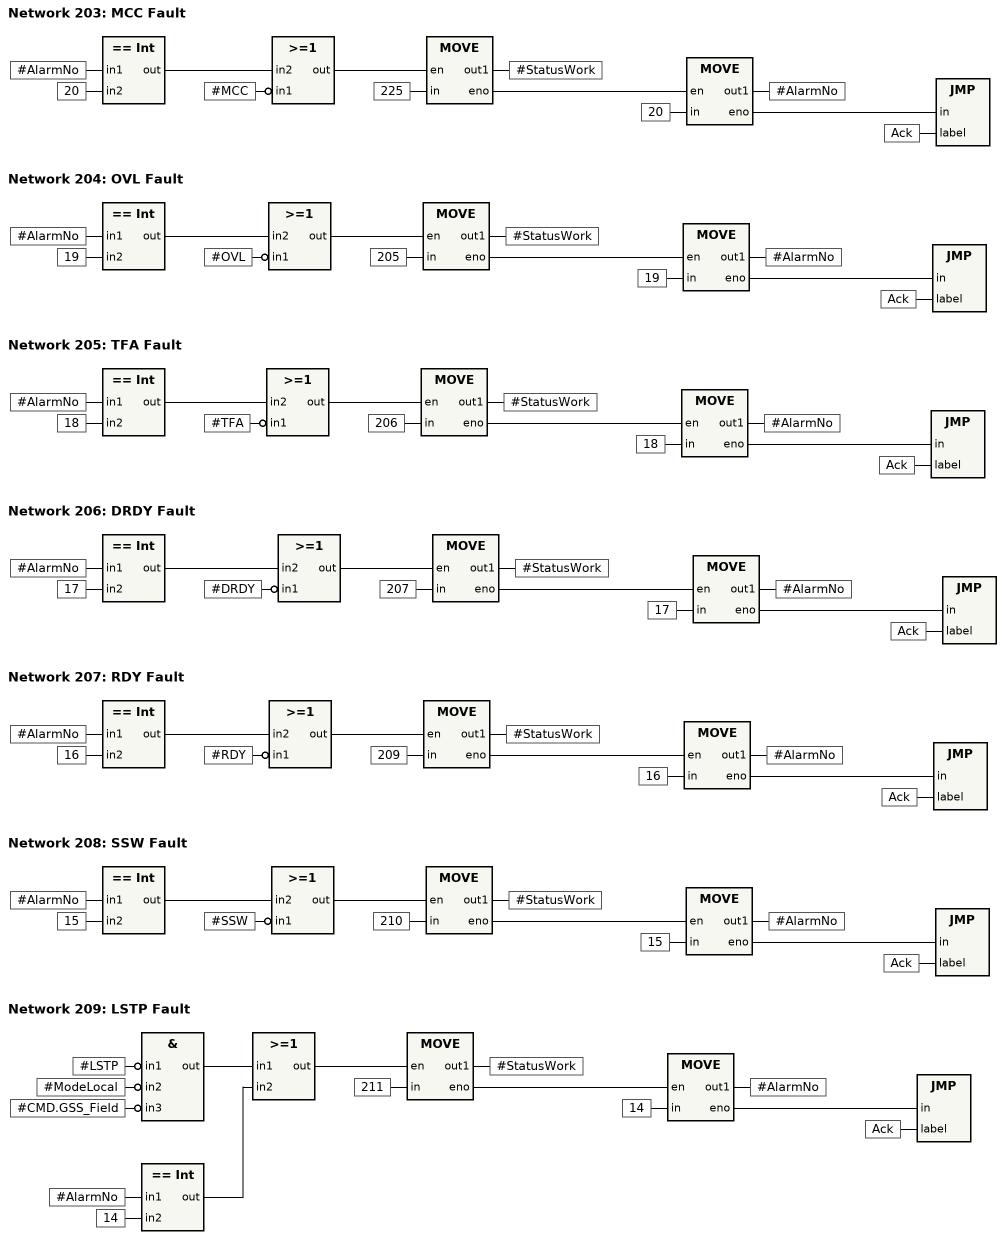
   // ENO of a box is taken as its EN; it also drops when the box reports an error
   #_w1 := (#AlarmNo = 20) OR NOT #MCC;
   IF #_w1 THEN
       #StatusWork := 225;
       #AlarmNo := 20;
       GOTO Ack;
   END_IF;
END_REGION

REGION Network 204: OVL Fault
   // ENO of a box is taken as its EN; it also drops when the box reports an error
   #_w1 := (#AlarmNo = 19) OR NOT #OVL;
   IF #_w1 THEN
       #StatusWork := 205;
       #AlarmNo := 19;
       GOTO Ack;
   END_IF;
END_REGION

REGION Network 205: TFA Fault
   // ENO of a box is taken as its EN; it also drops when the box reports an error
   #_w1 := (#AlarmNo = 18) OR NOT #TFA;
   IF #_w1 THEN
       #StatusWork := 206;
       #AlarmNo := 18;
       GOTO Ack;
   END_IF;
END_REGION

REGION Network 206: DRDY Fault
   // ENO of a box is taken as its EN; it also drops when the box reports an error
   #_w1 := (#AlarmNo = 17) OR NOT #DRDY;
   IF #_w1 THEN
       #StatusWork := 207;
       #AlarmNo := 17;
       GOTO Ack;
   END_IF;
END_REGION

REGION Network 207: RDY Fault
   // ENO of a box is taken as its EN; it also drops when the box reports an error
   #_w1 := (#AlarmNo = 16) OR NOT #RDY;
   IF #_w1 THEN
       #StatusWork := 209;
       #AlarmNo := 16;
       GOTO Ack;
   END_IF;
END_REGION

REGION Network 208: SSW Fault
   // ENO of a box is taken as its EN; it also drops when the box reports an error
   #_w1 := (#AlarmNo = 15) OR NOT #SSW;
   IF #_w1 THEN
       #StatusWork := 210;
       #AlarmNo := 15;
       GOTO Ack;
   END_IF;
END_REGION

REGION Network 209: LSTP Fault
   // ENO of a box is taken as its EN; it also drops when the box reports an error
   #_w1 := (NOT #LSTP AND NOT #ModeLocal AND NOT #CMD.GSS_Field) OR (#AlarmNo = 14);
   IF #_w1 THEN
       #StatusWork := 211;
       #AlarmNo := 14;
       GOTO Ack;
   END_IF;
END_REGION

REGION Network 210: REM Fault
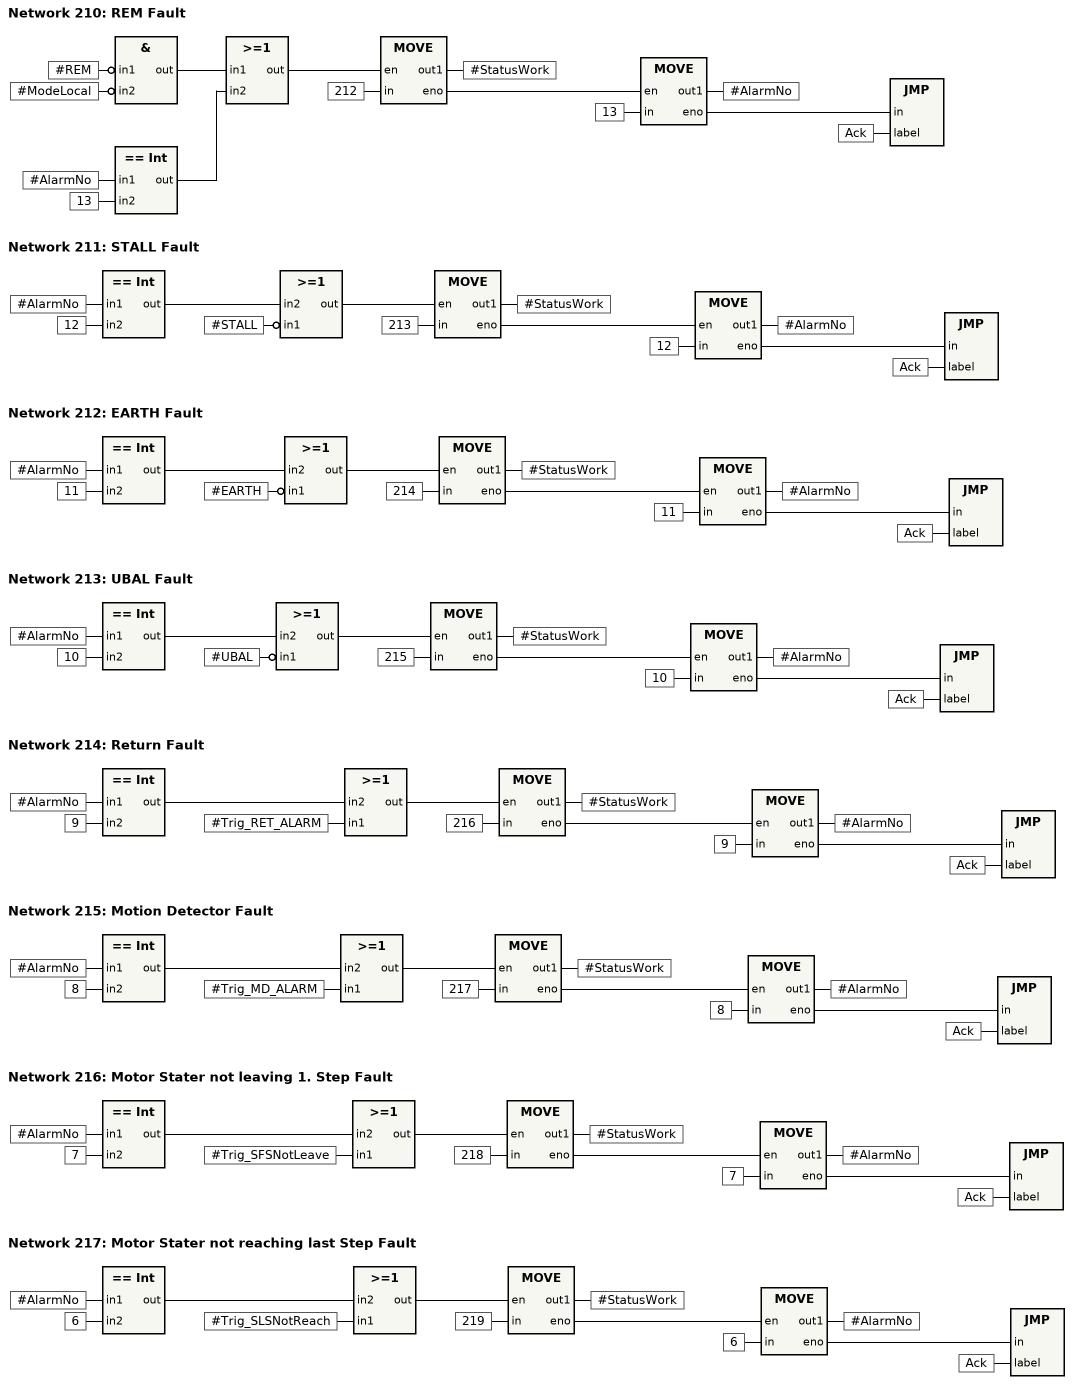
   // ENO of a box is taken as its EN; it also drops when the box reports an error
   #_w1 := (NOT #REM AND NOT #ModeLocal) OR (#AlarmNo = 13);
   IF #_w1 THEN
       #StatusWork := 212;
       #AlarmNo := 13;
       GOTO Ack;
   END_IF;
END_REGION

REGION Network 211: STALL Fault
   // ENO of a box is taken as its EN; it also drops when the box reports an error
   #_w1 := (#AlarmNo = 12) OR NOT #STALL;
   IF #_w1 THEN
       #StatusWork := 213;
       #AlarmNo := 12;
       GOTO Ack;
   END_IF;
END_REGION

REGION Network 212: EARTH Fault
   // ENO of a box is taken as its EN; it also drops when the box reports an error
   #_w1 := (#AlarmNo = 11) OR NOT #EARTH;
   IF #_w1 THEN
       #StatusWork := 214;
       #AlarmNo := 11;
       GOTO Ack;
   END_IF;
END_REGION

REGION Network 213: UBAL Fault
   // ENO of a box is taken as its EN; it also drops when the box reports an error
   #_w1 := (#AlarmNo = 10) OR NOT #UBAL;
   IF #_w1 THEN
       #StatusWork := 215;
       #AlarmNo := 10;
       GOTO Ack;
   END_IF;
END_REGION

REGION Network 214: Return Fault
   // ENO of a box is taken as its EN; it also drops when the box reports an error
   #_w1 := (#AlarmNo = 9) OR #Trig_RET_ALARM;
   IF #_w1 THEN
       #StatusWork := 216;
       #AlarmNo := 9;
       GOTO Ack;
   END_IF;
END_REGION

REGION Network 215: Motion Detector Fault
   // ENO of a box is taken as its EN; it also drops when the box reports an error
   #_w1 := (#AlarmNo = 8) OR #Trig_MD_ALARM;
   IF #_w1 THEN
       #StatusWork := 217;
       #AlarmNo := 8;
       GOTO Ack;
   END_IF;
END_REGION

REGION Network 216: Motor Stater not leaving 1. Step Fault
   // ENO of a box is taken as its EN; it also drops when the box reports an error
   #_w1 := (#AlarmNo = 7) OR #Trig_SFSNotLeave;
   IF #_w1 THEN
       #StatusWork := 218;
       #AlarmNo := 7;
       GOTO Ack;
   END_IF;
END_REGION

REGION Network 217: Motor Stater not reaching last Step Fault
   // ENO of a box is taken as its EN; it also drops when the box reports an error
   #_w1 := (#AlarmNo = 6) OR #Trig_SLSNotReach;
   IF #_w1 THEN
       #StatusWork := 219;
       #AlarmNo := 6;
       GOTO Ack;
   END_IF;
END_REGION

REGION Network 218: Motor Stater not reaching 1. Step Fault
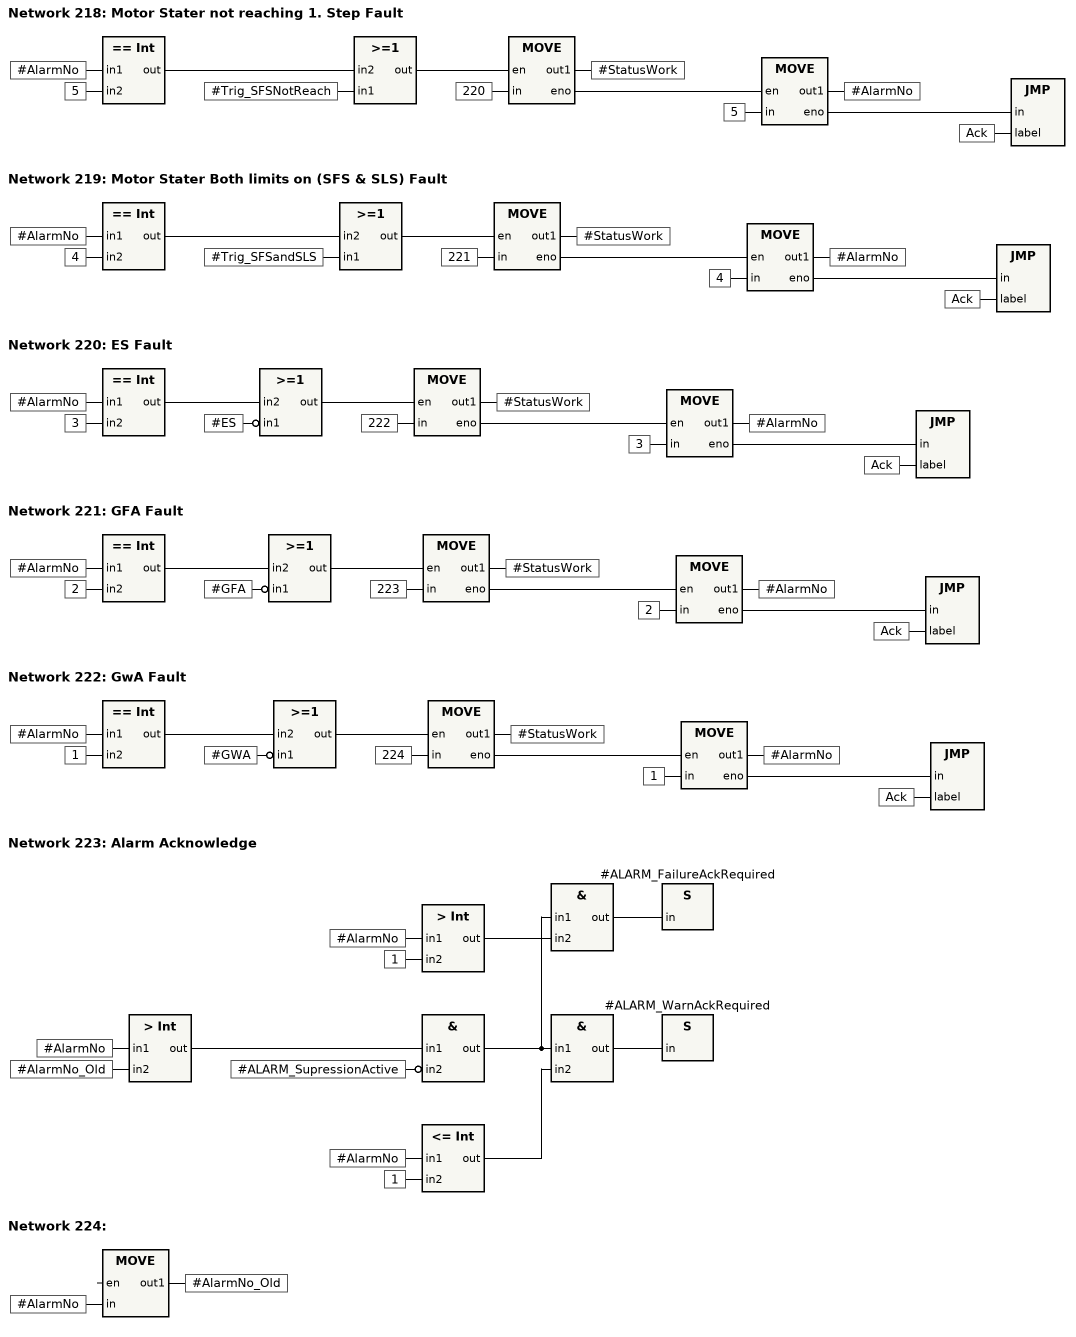
   // ENO of a box is taken as its EN; it also drops when the box reports an error
   #_w1 := (#AlarmNo = 5) OR #Trig_SFSNotReach;
   IF #_w1 THEN
       #StatusWork := 220;
       #AlarmNo := 5;
       GOTO Ack;
   END_IF;
END_REGION

REGION Network 219: Motor Stater Both limits on (SFS & SLS) Fault
   // ENO of a box is taken as its EN; it also drops when the box reports an error
   #_w1 := (#AlarmNo = 4) OR #Trig_SFSandSLS;
   IF #_w1 THEN
       #StatusWork := 221;
       #AlarmNo := 4;
       GOTO Ack;
   END_IF;
END_REGION

REGION Network 220: ES Fault
   // ENO of a box is taken as its EN; it also drops when the box reports an error
   #_w1 := (#AlarmNo = 3) OR NOT #ES;
   IF #_w1 THEN
       #StatusWork := 222;
       #AlarmNo := 3;
       GOTO Ack;
   END_IF;
END_REGION

REGION Network 221: GFA Fault
   // ENO of a box is taken as its EN; it also drops when the box reports an error
   #_w1 := (#AlarmNo = 2) OR NOT #GFA;
   IF #_w1 THEN
       #StatusWork := 223;
       #AlarmNo := 2;
       GOTO Ack;
   END_IF;
END_REGION

REGION Network 222: GwA Fault
   // ENO of a box is taken as its EN; it also drops when the box reports an error
   #_w1 := (#AlarmNo = 1) OR NOT #GWA;
   IF #_w1 THEN
       #StatusWork := 224;
       #AlarmNo := 1;
       GOTO Ack;
   END_IF;
END_REGION

REGION Network 223: Alarm Acknowledge
   Ack:
   #_w1 := (#AlarmNo > #AlarmNo_Old) AND NOT #ALARM_SupressionActive;
   IF #_w1 AND (#AlarmNo > 1) THEN #ALARM_FailureAckRequired := TRUE; END_IF;
   IF #_w1 AND (#AlarmNo <= 1) THEN #ALARM_WarnAckRequired := TRUE; END_IF;
END_REGION

REGION Network 224
   #AlarmNo_Old := #AlarmNo;
END_REGION

REGION Network 225
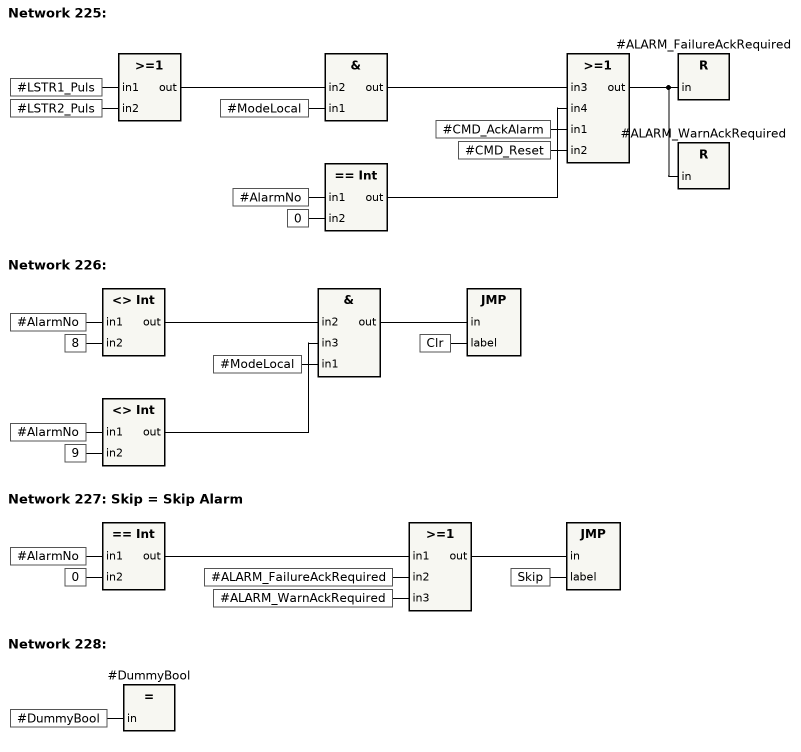
   IF ((#LSTR1_Puls OR #LSTR2_Puls) AND #ModeLocal) OR (#AlarmNo = 0) OR #CMD_AckAlarm OR #CMD_Reset THEN
       #ALARM_FailureAckRequired := FALSE;
       #ALARM_WarnAckRequired := FALSE;
   END_IF;
END_REGION

REGION Network 226
   IF (#AlarmNo <> 8) AND (#AlarmNo <> 9) AND #ModeLocal THEN GOTO Clr; END_IF;
END_REGION

REGION Network 227: Skip = Skip Alarm
   IF (#AlarmNo = 0) OR #ALARM_FailureAckRequired OR #ALARM_WarnAckRequired THEN GOTO Skip; END_IF;
END_REGION

REGION Network 228
   Clr:
   #DummyBool := #DummyBool;
END_REGION

REGION Network 229
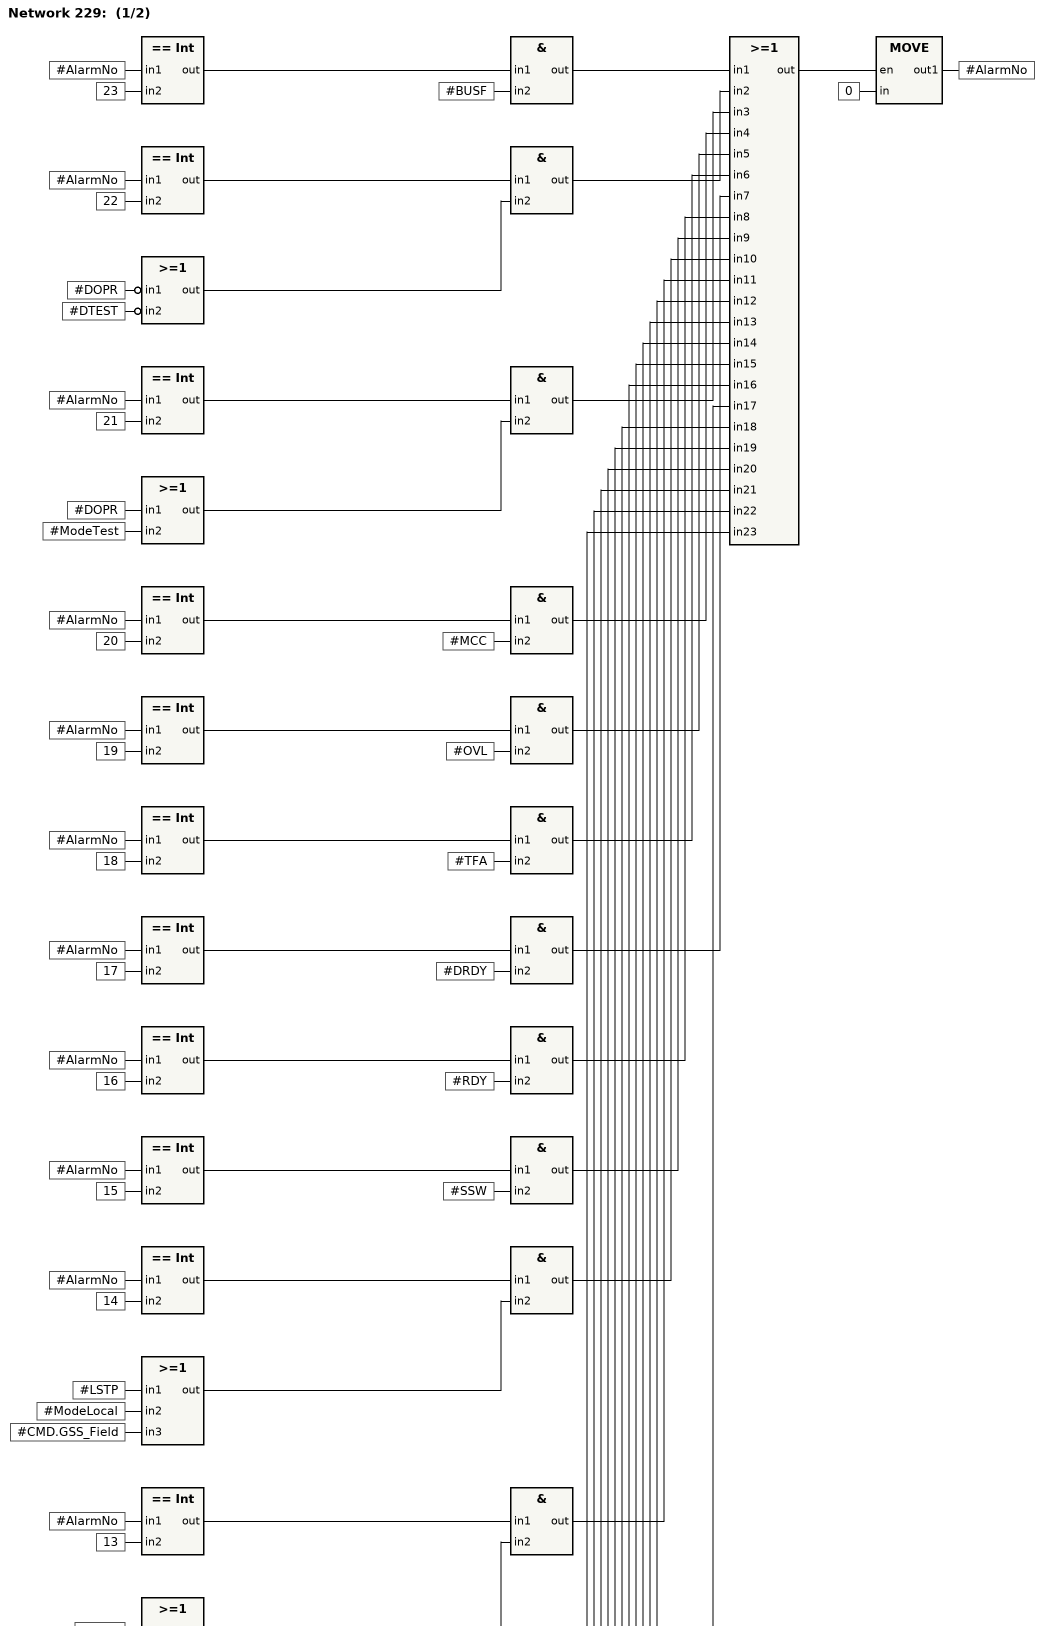
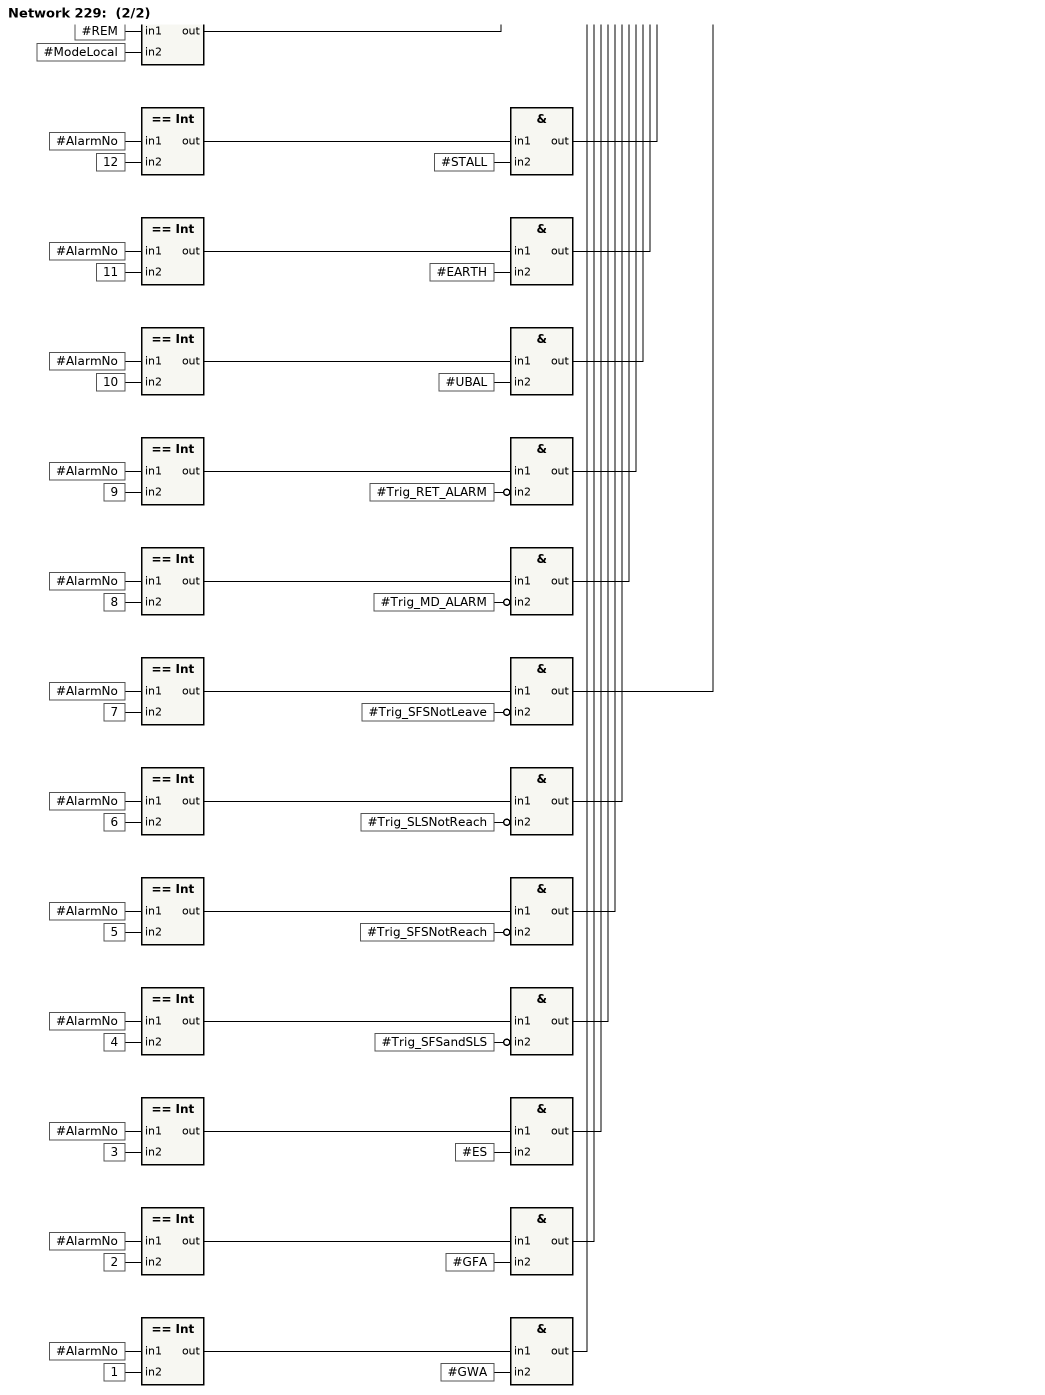
   IF ((#AlarmNo = 23) AND #BUSF) OR ((#AlarmNo = 22) AND (NOT #DOPR OR NOT #DTEST)) OR ((#AlarmNo = 21) AND (#DOPR OR #ModeTest)) OR ((#AlarmNo = 20) AND #MCC) OR ((#AlarmNo = 19) AND #OVL) OR ((#AlarmNo = 18) AND #TFA) OR ((#AlarmNo = 17) AND #DRDY) OR ((#AlarmNo = 16) AND #RDY) OR ((#AlarmNo = 15) AND #SSW) OR ((#AlarmNo = 14) AND (#LSTP OR #ModeLocal OR #CMD.GSS_Field)) OR ((#AlarmNo = 13) AND (#REM OR #ModeLocal)) OR ((#AlarmNo = 12) AND #STALL) OR ((#AlarmNo = 11) AND #EARTH) OR ((#AlarmNo = 10) AND #UBAL) OR ((#AlarmNo = 9) AND NOT #Trig_RET_ALARM) OR ((#AlarmNo = 8) AND NOT #Trig_MD_ALARM) OR ((#AlarmNo = 7) AND NOT #Trig_SFSNotLeave) OR ((#AlarmNo = 6) AND NOT #Trig_SLSNotReach) OR ((#AlarmNo = 5) AND NOT #Trig_SFSNotReach) OR ((#AlarmNo = 4) AND NOT #Trig_SFSandSLS) OR ((#AlarmNo = 3) AND #ES) OR ((#AlarmNo = 2) AND #GFA) OR ((#AlarmNo = 1) AND #GWA) THEN
       #AlarmNo := 0;
   END_IF;
END_REGION

REGION Network 230
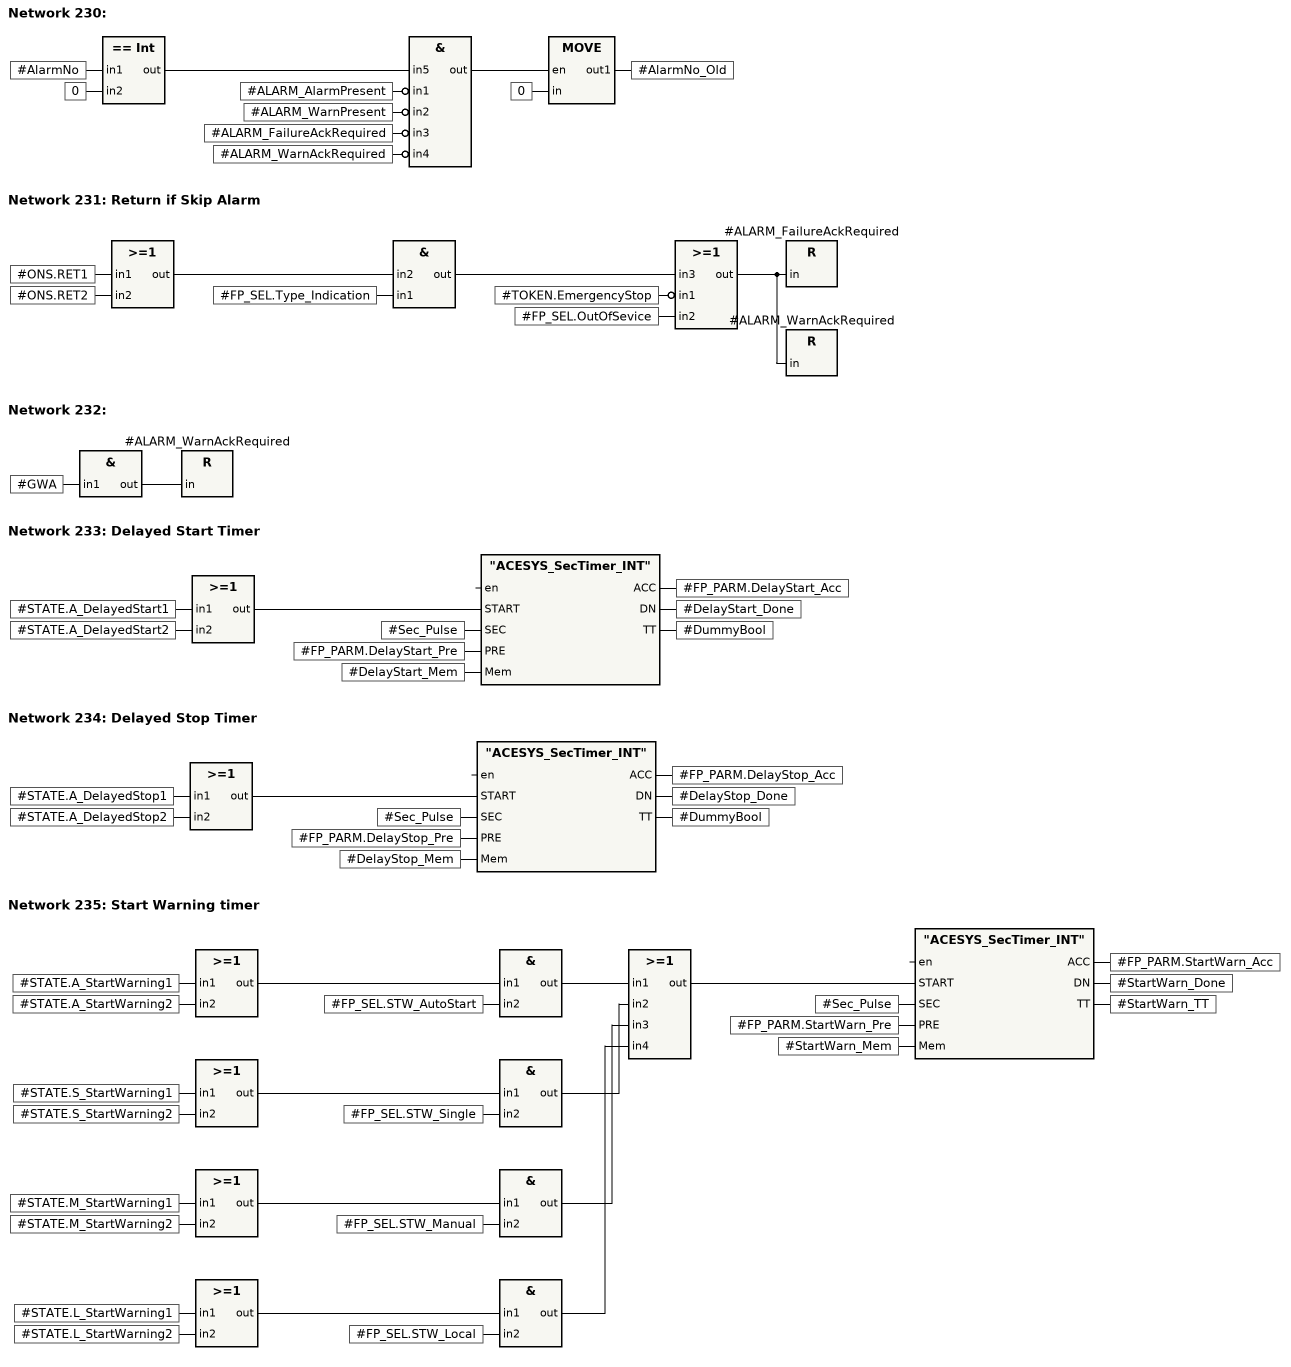
   IF (#AlarmNo = 0) AND NOT #ALARM_AlarmPresent AND NOT #ALARM_WarnPresent AND NOT #ALARM_FailureAckRequired AND NOT #ALARM_WarnAckRequired THEN
       #AlarmNo_Old := 0;
   END_IF;
END_REGION

REGION Network 231: Return if Skip Alarm
   // Alarm/Warning are Auto Acknowledged on EmergencyStop
   // Build 002 - 25 March 2019 : Alarm/Warning are Auto Acknowledged on OutOfService
   // Build 003 - 30 June 2019 (EXTBOB): Acknowledge pending alarms when Unit started as "Indication"
   Skip:
   IF ((#ONS.RET1 OR #ONS.RET2) AND #FP_SEL.Type_Indication) OR NOT #TOKEN.EmergencyStop OR #FP_SEL.OutOfSevice THEN
       #ALARM_FailureAckRequired := FALSE;
       #ALARM_WarnAckRequired := FALSE;
   END_IF;
END_REGION

REGION Network 232
   // Build 005 - 30.July.2019 (MIA-US): General Warning status is "auto-reset" in ECS (clears without an acknowledge).  "ALARM_WarnAckRequired" flag should also be reset to allow clearing of the AlarmNo register.
   IF #GWA THEN #ALARM_WarnAckRequired := FALSE; END_IF;
END_REGION

REGION Network 233: Delayed Start Timer
   "ACESYS_SecTimer_INT"(START := #STATE.A_DelayedStart1 OR #STATE.A_DelayedStart2,
                         SEC := #Sec_Pulse,
                         PRE := #FP_PARM.DelayStart_Pre,
                         Mem := #DelayStart_Mem,
                         ACC => #FP_PARM.DelayStart_Acc,
                         DN => #DelayStart_Done,
                         TT => #DummyBool);
END_REGION

REGION Network 234: Delayed Stop Timer
   "ACESYS_SecTimer_INT"(START := #STATE.A_DelayedStop1 OR #STATE.A_DelayedStop2,
                         SEC := #Sec_Pulse,
                         PRE := #FP_PARM.DelayStop_Pre,
                         Mem := #DelayStop_Mem,
                         ACC => #FP_PARM.DelayStop_Acc,
                         DN => #DelayStop_Done,
                         TT => #DummyBool);
END_REGION

REGION Network 235: Start Warning timer
   // Build 003 - 30 June 2019 (EXTBOB) : Added STW selection to avoid ASTW pulse
   "ACESYS_SecTimer_INT"(START := ((#STATE.A_StartWarning1 OR #STATE.A_StartWarning2) AND #FP_SEL.STW_AutoStart) OR ((#STATE.S_StartWarning1 OR #STATE.S_StartWarning2) AND #FP_SEL.STW_Single) OR ((#STATE.M_StartWarning1 OR #STATE.M_StartWarning2) AND #FP_SEL.STW_Manual) OR ((#STATE.L_StartWarning1 OR #STATE.L_StartWarning2) AND #FP_SEL.STW_Local),
                         SEC := #Sec_Pulse,
                         PRE := #FP_PARM.StartWarn_Pre,
                         Mem := #StartWarn_Mem,
                         ACC => #FP_PARM.StartWarn_Acc,
                         DN => #StartWarn_Done,
                         TT => #StartWarn_TT);
END_REGION

REGION Network 236: Run Delay 1 Timer
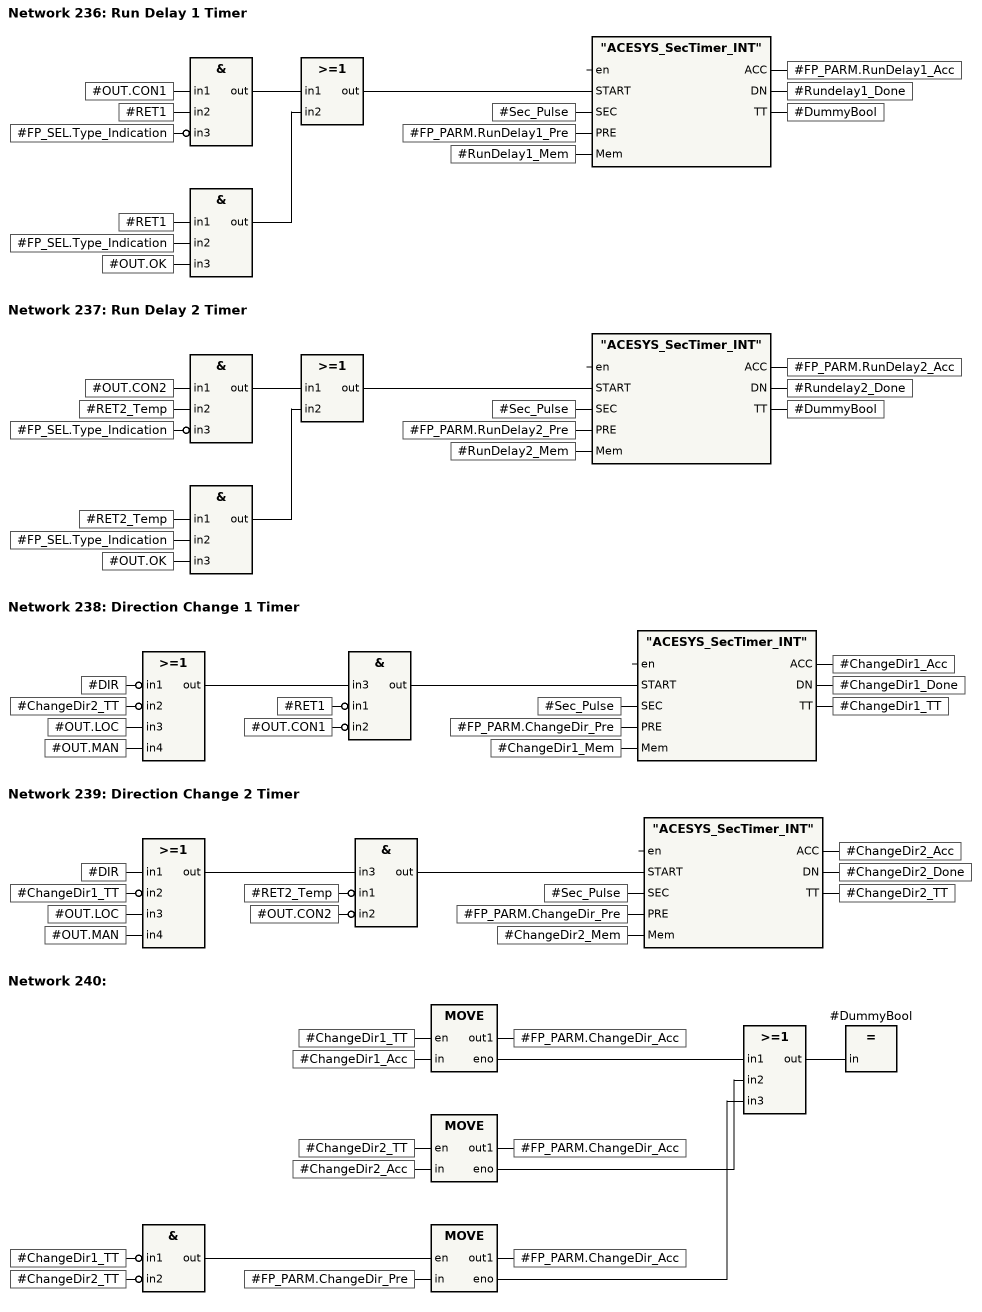
   "ACESYS_SecTimer_INT"(START := (#OUT.CON1 AND #RET1 AND NOT #FP_SEL.Type_Indication) OR (#RET1 AND #FP_SEL.Type_Indication AND #OUT.OK),
                         SEC := #Sec_Pulse,
                         PRE := #FP_PARM.RunDelay1_Pre,
                         Mem := #RunDelay1_Mem,
                         ACC => #FP_PARM.RunDelay1_Acc,
                         DN => #Rundelay1_Done,
                         TT => #DummyBool);
END_REGION

REGION Network 237: Run Delay 2 Timer
   "ACESYS_SecTimer_INT"(START := (#OUT.CON2 AND #RET2_Temp AND NOT #FP_SEL.Type_Indication) OR (#RET2_Temp AND #FP_SEL.Type_Indication AND #OUT.OK),
                         SEC := #Sec_Pulse,
                         PRE := #FP_PARM.RunDelay2_Pre,
                         Mem := #RunDelay2_Mem,
                         ACC => #FP_PARM.RunDelay2_Acc,
                         DN => #Rundelay2_Done,
                         TT => #DummyBool);
END_REGION

REGION Network 238: Direction Change 1 Timer
   // Build 007 - 03. Dec 2019 (EXTBOB) : DIR Neg logic, CON1 Neg flag added series to activate this timer during direction change at starting when return signal is 0
   "ACESYS_SecTimer_INT"(START := (NOT #DIR OR NOT #ChangeDir2_TT OR #OUT.LOC OR #OUT.MAN) AND NOT #RET1 AND NOT #OUT.CON1,
                         SEC := #Sec_Pulse,
                         PRE := #FP_PARM.ChangeDir_Pre,
                         Mem := #ChangeDir1_Mem,
                         ACC => #ChangeDir1_Acc,
                         DN => #ChangeDir1_Done,
                         TT => #ChangeDir1_TT);
END_REGION

REGION Network 239: Direction Change 2 Timer
   // Build 007 - 03. Dec 2019 (EXTBOB) : DIR  logic, CON2 Neg flag added series to activate this timer during direction change at starting when return signal is 0
   "ACESYS_SecTimer_INT"(START := (#DIR OR NOT #ChangeDir1_TT OR #OUT.LOC OR #OUT.MAN) AND NOT #RET2_Temp AND NOT #OUT.CON2,
                         SEC := #Sec_Pulse,
                         PRE := #FP_PARM.ChangeDir_Pre,
                         Mem := #ChangeDir2_Mem,
                         ACC => #ChangeDir2_Acc,
                         DN => #ChangeDir2_Done,
                         TT => #ChangeDir2_TT);
END_REGION

REGION Network 240
   // ENO of a box is taken as its EN; it also drops when the box reports an error
   IF #ChangeDir1_TT THEN #FP_PARM.ChangeDir_Acc := #ChangeDir1_Acc; END_IF;
   IF #ChangeDir2_TT THEN #FP_PARM.ChangeDir_Acc := #ChangeDir2_Acc; END_IF;
   #_w1 := NOT #ChangeDir1_TT AND NOT #ChangeDir2_TT;
   IF #_w1 THEN #FP_PARM.ChangeDir_Acc := #FP_PARM.ChangeDir_Pre; END_IF;
   #DummyBool := #ChangeDir1_TT OR #ChangeDir2_TT OR #_w1;
END_REGION

REGION Network 241: Rotor Starter: Leaving first Step Timer
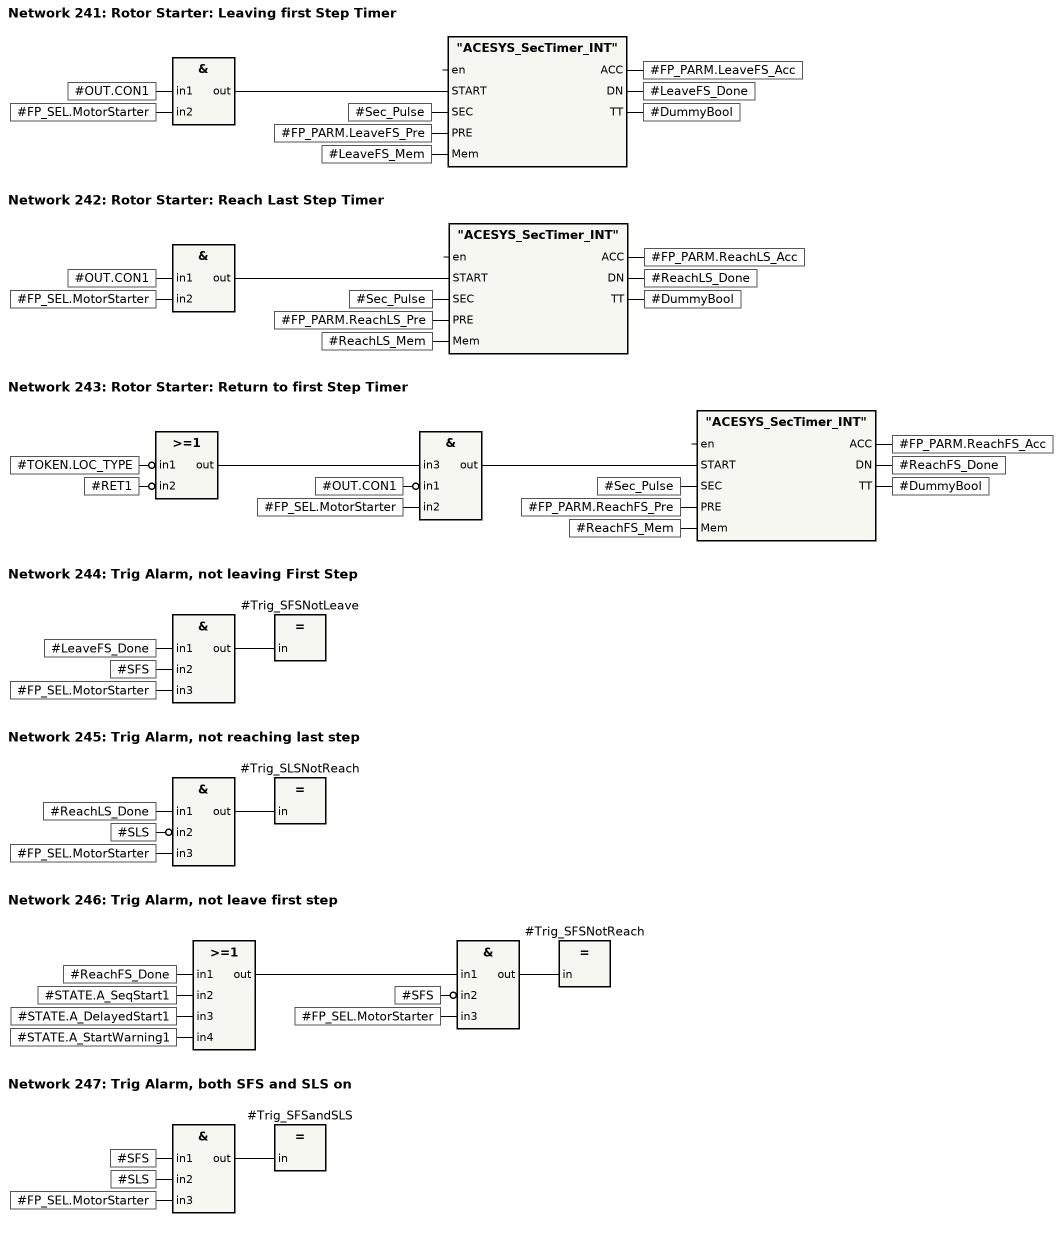
   "ACESYS_SecTimer_INT"(START := #OUT.CON1 AND #FP_SEL.MotorStarter,
                         SEC := #Sec_Pulse,
                         PRE := #FP_PARM.LeaveFS_Pre,
                         Mem := #LeaveFS_Mem,
                         ACC => #FP_PARM.LeaveFS_Acc,
                         DN => #LeaveFS_Done,
                         TT => #DummyBool);
END_REGION

REGION Network 242: Rotor Starter: Reach Last Step Timer
   "ACESYS_SecTimer_INT"(START := #OUT.CON1 AND #FP_SEL.MotorStarter,
                         SEC := #Sec_Pulse,
                         PRE := #FP_PARM.ReachLS_Pre,
                         Mem := #ReachLS_Mem,
                         ACC => #FP_PARM.ReachLS_Acc,
                         DN => #ReachLS_Done,
                         TT => #DummyBool);
END_REGION

REGION Network 243: Rotor Starter: Return to first Step Timer
   // Build 003 - 1.July.2019 (EXTBOB): Added logic to inhibit starter fault when running in "electrical" local mode.
   "ACESYS_SecTimer_INT"(START := (NOT #TOKEN.LOC_TYPE OR NOT #RET1) AND NOT #OUT.CON1 AND #FP_SEL.MotorStarter,
                         SEC := #Sec_Pulse,
                         PRE := #FP_PARM.ReachFS_Pre,
                         Mem := #ReachFS_Mem,
                         ACC => #FP_PARM.ReachFS_Acc,
                         DN => #ReachFS_Done,
                         TT => #DummyBool);
END_REGION

REGION Network 244: Trig Alarm, not leaving First Step
   #Trig_SFSNotLeave := #LeaveFS_Done AND #SFS AND #FP_SEL.MotorStarter;
END_REGION

REGION Network 245: Trig Alarm, not reaching last step
   #Trig_SLSNotReach := #ReachLS_Done AND NOT #SLS AND #FP_SEL.MotorStarter;
END_REGION

REGION Network 246: Trig Alarm, not leave first step
   // Build 029 - 23.Sep.2021 (SURAM-IN) : A_Selected is replaced with A_SeqStart1 or A_DelayedStart1 or A_StartWarning1
   #Trig_SFSNotReach := (#ReachFS_Done OR #STATE.A_SeqStart1 OR #STATE.A_DelayedStart1 OR #STATE.A_StartWarning1) AND NOT #SFS AND #FP_SEL.MotorStarter;
END_REGION

REGION Network 247: Trig Alarm, both SFS and SLS on
   #Trig_SFSandSLS := #SFS AND #SLS AND #FP_SEL.MotorStarter;
END_REGION

REGION Network 248: Return Monitoring Fault
